// TIA Portal V16 export
// export: Created 2021-11-12T13:32:21.9335277Z, ExportSetting WithDefaults, DisplayName Totally Integrated Automation Portal, DisplayVersion V16 Update 3, DisplayName TIA Portal Version Control Interface, DisplayVersion V16 Update 2, DisplayName TIA Portal Openness, DisplayVersion V16 Update 3, DisplayName SINAMICS Startdrive Advanced, DisplayVersion V16 Update 5, DisplayName SINAMICS Startdrive G130, G150, S120, S150, SINAMICS MV, S210, DisplayVersion V16 Update 5, DisplayName SINAMICS Startdrive G110M, G120, G120C, G120D, G120P, G115D, DisplayVersion V16 Update 5, DisplayName STEP 7 Professional, DisplayVersion V16 Update 3, DisplayName STEP 7 Safety, DisplayVersion V16, DisplayName WinCC UA Professional, DisplayVersion V16 Update 3
FUNCTION_BLOCK "Station1R2"   // FB34, LAD
{ S7_Optimized_Access := 'TRUE' }
VERSION : 0.1
// stored: AutoNumber true, IsIECCheckEnabled false, IsRetainMemResEnabled false, MemoryReserve 100, SetENOAutomatically false, UDAEnableTagReadback false
   VAR
      SF_RO01_Timeout : "STD_DI_Mon";   // Move timeout
      "SF_CL01-BG01_Alarm" { S7_SetPoint := 'True'} : "STD_DI_Mon";
      "SF_CL01-BG02_Alarm" { S7_SetPoint := 'True'} : "STD_DI_Mon";
      SF_RC01 : "STD_DriveRobotABB";
      SF_RO01 : "STD_RobotABB";
      SF_RobotGripper : "STD_RobotGripper";
      SS_RobotZones { S7_SetPoint := 'True'} : "STD_RobotZones";
      SS_Edge { S7_SetPoint := 'True'} : Array[0..100] of Bool;
   END_VAR
   VAR RETAIN
      SDIPartID : DInt;
      SI_PartType : Int;
   END_VAR
   VAR
      SI_140RowNo : Int;   // Row number in map of station 140
      SI_140LineNo : Int;   // Line number in map of station 140
      SB1PutPosFound140 : Bool;   // Put position in map of station 140 found
      SB1ReqToChangeTool : Bool;   // Request from zone command to change tools
      SB1_1R2ChangeToolDone : Bool;   // Changing tool process done
      SB1_1R2GripperToTakeUp : Bool;
      SB1_1R2PutToolDone : Bool;
      SB1_1R1ToolSwitchDone : Bool;
      SB1CycleAutostop : Bool;   // Cycle autostop command
      SB1ServicePosReq { ExternalAccessible := 'False'; ExternalVisible := 'False'; ExternalWritable := 'False'} : Bool;   // Request to go to/from service position
      SB1RobotInitialized : Bool;   // Robot is initialized
   END_VAR
   VAR_TEMP
      TS_RC01 : "UDT_DriveRobotABBControl";   // Robot controller RC01 control
      TS_RO01 : "UDT_RobotABBControl";   // Robot RO01 control
      TI_RowNo : Int;
      TI_LineNo : Int;
      TB1PwrOK : Bool;   // Power for this station is OK
      TB1HomePosReq : Bool;   // Request to go to home position
      TB1Take120 : Bool;   // Take parts from 120
      TB1Put140 : Bool;   // Put parts to 140
      TB1CtrlRun : Bool;   // Robot controller is running in automat
      TB1GripperFree : Bool;
      TB1ChangeTool1R1UpDown : Bool;   // Change tool from upper possition
      TB1ChangeTool1R1DownUp : Bool;   // Change tool from lower possition
      TB1PutTool1R2Up : Bool;
      TB1PutTool1R2Down : Bool;
      TB1TakeTool1R2Up : Bool;
      TB1TakeTool1R2Down : Bool;
   END_VAR
   VAR CONSTANT
      CI_JobHome : UInt := 1;
      CI_JobService : UInt := 2;
      CI_JobPutToo1R2Up : UInt := 11;
      CI_JobPutToo1R2Down : UInt := 12;
      CI_JobChangeTool1R1UpDown : UInt := 21;
      CI_JobChangeTool1R1DownUp : UInt := 22;
      CI_JobTakeTool1R2Up : UInt := 31;
      CI_JobTakeTool1R2Down : UInt := 32;
      CI_JobTakeParts : UInt := 100;
      CI_JobPutPartsPos11 : UInt := 201;
      CI_JobPutPartsPos15 : UInt := 202;
      CI_JobPutPartsPos19 : UInt := 203;
      CI_JobPutPartsPos21 : UInt := 204;
      CI_JobPutPartsPos25 : UInt := 205;
      CI_JobPutPartsPos29 : UInt := 206;
   END_VAR
   VAR_TEMP   // added for the SCL form of the ladder/FBD networks
      _w1 : Bool;
      _w2 : Bool;
      _w3 : Bool;
      _w4 : Bool;
      _w5 : Bool;
      _w6 : Bool;
      _w7 : Bool;
      _w8 : Bool;
   END_VAR
BEGIN

REGION Network 1: Clear temporary variables
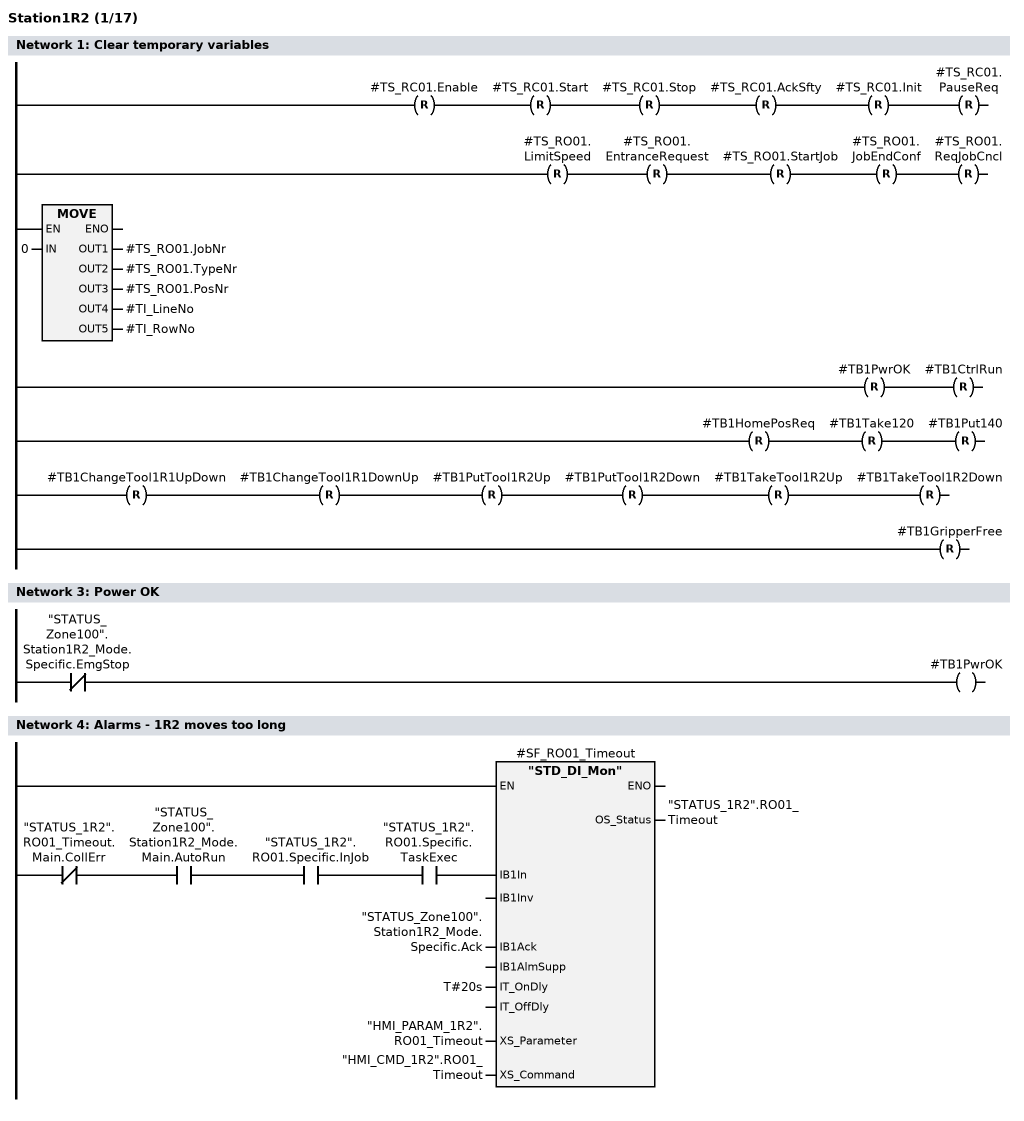
   RUNG wire#powerrail
      R_Coil( #TS_RC01.Enable )
      R_Coil( #TS_RC01.Start )
      R_Coil( #TS_RC01.Stop )
      R_Coil( #TS_RC01.AckSfty )
      R_Coil( #TS_RC01.Init )
      R_Coil( #TS_RC01.PauseReq )
   END_RUNG
   RUNG wire#powerrail
      R_Coil( #TS_RO01.LimitSpeed )
      R_Coil( #TS_RO01.EntranceRequest )
      R_Coil( #TS_RO01.StartJob )
      R_Coil( #TS_RO01.JobEndConf )
      R_Coil( #TS_RO01.ReqJobCncl )
   END_RUNG
   RUNG wire#powerrail
      Move(in := 0, out1 => #TS_RO01.JobNr, out2 => #TS_RO01.TypeNr, out3 => #TS_RO01.PosNr, out4 => #TI_LineNo, out5 => #TI_RowNo)
   END_RUNG
   RUNG wire#powerrail
      R_Coil( #TB1PwrOK )
      R_Coil( #TB1CtrlRun )
   END_RUNG
   RUNG wire#powerrail
      R_Coil( #TB1HomePosReq )
      R_Coil( #TB1Take120 )
      R_Coil( #TB1Put140 )
   END_RUNG
   RUNG wire#powerrail
      R_Coil( #TB1ChangeTool1R1UpDown )
      R_Coil( #TB1ChangeTool1R1DownUp )
      R_Coil( #TB1PutTool1R2Up )
      R_Coil( #TB1PutTool1R2Down )
      R_Coil( #TB1TakeTool1R2Up )
      R_Coil( #TB1TakeTool1R2Down )
   END_RUNG
   RUNG wire#powerrail
      R_Coil( #TB1GripperFree )
   END_RUNG
   // the same network as SCL:
   #TS_RC01.Enable := FALSE;
   #TS_RC01.Start := FALSE;
   #TS_RC01.Stop := FALSE;
   #TS_RC01.AckSfty := FALSE;
   #TS_RC01.Init := FALSE;
   #TS_RC01.PauseReq := FALSE;
   #TS_RO01.LimitSpeed := FALSE;
   #TS_RO01.EntranceRequest := FALSE;
   #TS_RO01.StartJob := FALSE;
   #TS_RO01.JobEndConf := FALSE;
   #TS_RO01.ReqJobCncl := FALSE;
   #TS_RO01.JobNr := 0;
   #TS_RO01.TypeNr := 0;
   #TS_RO01.PosNr := 0;
   #TI_LineNo := 0;
   #TI_RowNo := 0;
   #TB1PwrOK := FALSE;
   #TB1CtrlRun := FALSE;
   #TB1HomePosReq := FALSE;
   #TB1Take120 := FALSE;
   #TB1Put140 := FALSE;
   #TB1ChangeTool1R1UpDown := FALSE;
   #TB1ChangeTool1R1DownUp := FALSE;
   #TB1PutTool1R2Up := FALSE;
   #TB1PutTool1R2Down := FALSE;
   #TB1TakeTool1R2Up := FALSE;
   #TB1TakeTool1R2Down := FALSE;
   #TB1GripperFree := FALSE;
END_REGION

REGION Network 2: *************** Alarms ***************
END_REGION

REGION Network 3: Power OK
   RUNG wire#powerrail
      I_Contact( "STATUS_Zone100".Station1R2_Mode.Specific.EmgStop )
      Coil( #TB1PwrOK )
   END_RUNG
   // the same network as SCL:
   #TB1PwrOK := NOT "STATUS_Zone100".Station1R2_Mode.Specific.EmgStop;
END_REGION

REGION Network 4: Alarms - 1R2 moves too long
   RUNG wire#powerrail
      #SF_RO01_Timeout(IB1In := wire#w1, IB1Inv :=, IB1Ack := "STATUS_Zone100".Station1R2_Mode.Specific.Ack, IB1AlmSupp :=, IT_OnDly := T#20s, IT_OffDly :=, XS_Parameter := "HMI_PARAM_1R2".RO01_Timeout, XS_Command := "HMI_CMD_1R2".RO01_Timeout, OS_Status => "STATUS_1R2".RO01_Timeout)
   END_RUNG
   RUNG wire#powerrail
      I_Contact( "STATUS_1R2".RO01_Timeout.Main.CollErr )
      Contact( "STATUS_Zone100".Station1R2_Mode.Main.AutoRun )
      Contact( "STATUS_1R2".RO01.Specific.InJob )
      Contact( "STATUS_1R2".RO01.Specific.TaskExec )
   END_RUNG wire#w1
   // the same network as SCL:
   #SF_RO01_Timeout(IB1In := NOT "STATUS_1R2".RO01_Timeout.Main.CollErr AND "STATUS_Zone100".Station1R2_Mode.Main.AutoRun AND "STATUS_1R2".RO01.Specific.InJob AND "STATUS_1R2".RO01.Specific.TaskExec,   // "STD_DI_Mon"
                    IB1Ack := "STATUS_Zone100".Station1R2_Mode.Specific.Ack,
                    IT_OnDly := T#20s,
                    XS_Parameter := "HMI_PARAM_1R2".RO01_Timeout,
                    XS_Command := "HMI_CMD_1R2".RO01_Timeout,
                    OS_Status => "STATUS_1R2".RO01_Timeout);
END_REGION

REGION Network 5: Sensor alarms - CL01
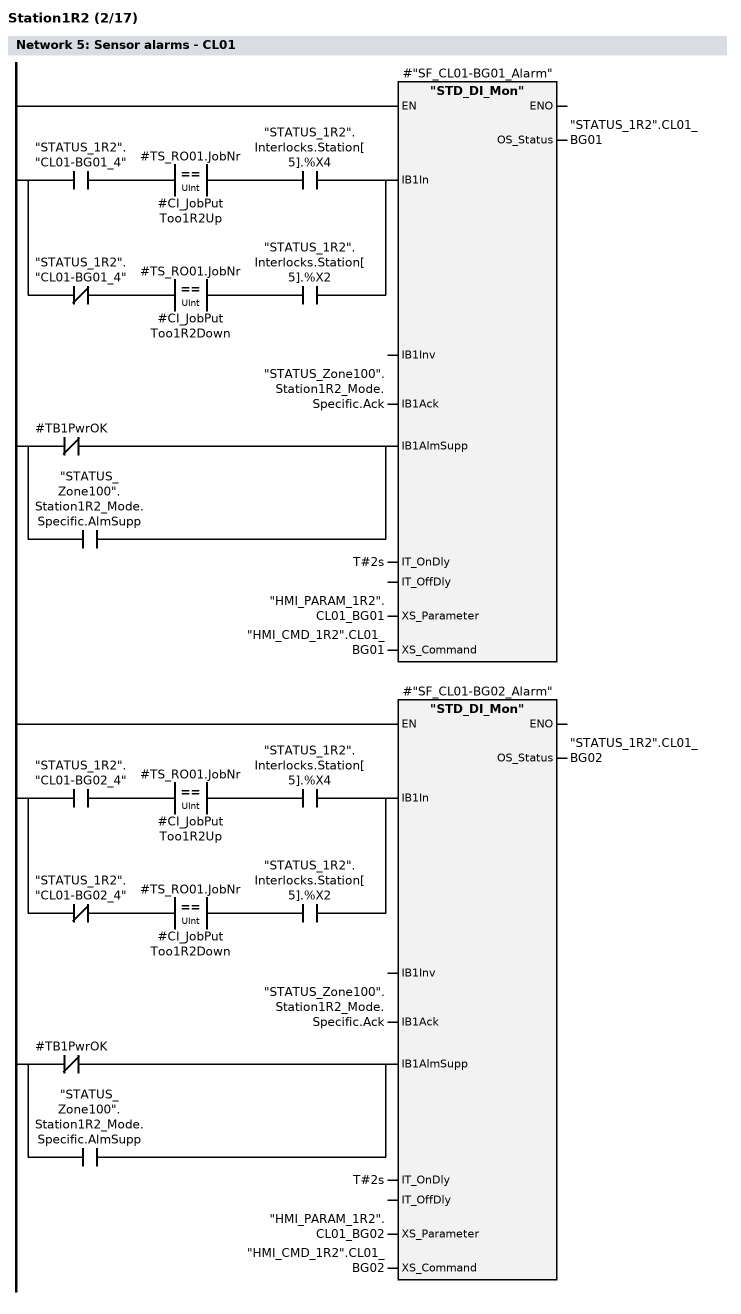
   RUNG wire#powerrail
      #"SF_CL01-BG01_Alarm"(IB1In := wire#w1, IB1AlmSupp := wire#w2, IB1Inv :=, IB1Ack := "STATUS_Zone100".Station1R2_Mode.Specific.Ack, IT_OnDly := T#2s, IT_OffDly :=, XS_Parameter := "HMI_PARAM_1R2".CL01_BG01, XS_Command := "HMI_CMD_1R2".CL01_BG01, OS_Status => "STATUS_1R2".CL01_BG01)
   END_RUNG
   RUNG wire#powerrail
      Contact( "STATUS_1R2"."CL01-BG01_4" )
      { S7_Templates := "SrcType := UInt" } EQ_Contact(in1 := #TS_RO01.JobNr, in2 := #CI_JobPutToo1R2Up)
      Contact( "STATUS_1R2".Interlocks.Station[5].%X4 )
   END_RUNG wire#w1
   RUNG wire#powerrail
      I_Contact( "STATUS_1R2"."CL01-BG01_4" )
      { S7_Templates := "SrcType := UInt" } EQ_Contact(in1 := #TS_RO01.JobNr, in2 := #CI_JobPutToo1R2Down)
      Contact( "STATUS_1R2".Interlocks.Station[5].%X2 )
   END_RUNG wire#w1
   RUNG wire#powerrail
      I_Contact( #TB1PwrOK )
   END_RUNG wire#w2
   RUNG wire#powerrail
      Contact( "STATUS_Zone100".Station1R2_Mode.Specific.AlmSupp )
   END_RUNG wire#w2
   RUNG wire#powerrail
      #"SF_CL01-BG02_Alarm"(IB1In := wire#w3, IB1AlmSupp := wire#w4, IB1Inv :=, IB1Ack := "STATUS_Zone100".Station1R2_Mode.Specific.Ack, IT_OnDly := T#2s, IT_OffDly :=, XS_Parameter := "HMI_PARAM_1R2".CL01_BG02, XS_Command := "HMI_CMD_1R2".CL01_BG02, OS_Status => "STATUS_1R2".CL01_BG02)
   END_RUNG
   RUNG wire#powerrail
      Contact( "STATUS_1R2"."CL01-BG02_4" )
      { S7_Templates := "SrcType := UInt" } EQ_Contact(in1 := #TS_RO01.JobNr, in2 := #CI_JobPutToo1R2Up)
      Contact( "STATUS_1R2".Interlocks.Station[5].%X4 )
   END_RUNG wire#w3
   RUNG wire#powerrail
      I_Contact( "STATUS_1R2"."CL01-BG02_4" )
      { S7_Templates := "SrcType := UInt" } EQ_Contact(in1 := #TS_RO01.JobNr, in2 := #CI_JobPutToo1R2Down)
      Contact( "STATUS_1R2".Interlocks.Station[5].%X2 )
   END_RUNG wire#w3
   RUNG wire#powerrail
      I_Contact( #TB1PwrOK )
   END_RUNG wire#w4
   RUNG wire#powerrail
      Contact( "STATUS_Zone100".Station1R2_Mode.Specific.AlmSupp )
   END_RUNG wire#w4
   // the same network as SCL:
   #"SF_CL01-BG01_Alarm"(IB1In := ("STATUS_1R2"."CL01-BG01_4" AND (#TS_RO01.JobNr = #CI_JobPutToo1R2Up) AND "STATUS_1R2".Interlocks.Station[5].%X4) OR (NOT "STATUS_1R2"."CL01-BG01_4" AND (#TS_RO01.JobNr = #CI_JobPutToo1R2Down) AND "STATUS_1R2".Interlocks.Station[5].%X2),   // "STD_DI_Mon"
                         IB1Ack := "STATUS_Zone100".Station1R2_Mode.Specific.Ack,
                         IB1AlmSupp := NOT #TB1PwrOK OR "STATUS_Zone100".Station1R2_Mode.Specific.AlmSupp,
                         IT_OnDly := T#2s,
                         XS_Parameter := "HMI_PARAM_1R2".CL01_BG01,
                         XS_Command := "HMI_CMD_1R2".CL01_BG01,
                         OS_Status => "STATUS_1R2".CL01_BG01);
   #"SF_CL01-BG02_Alarm"(IB1In := ("STATUS_1R2"."CL01-BG02_4" AND (#TS_RO01.JobNr = #CI_JobPutToo1R2Up) AND "STATUS_1R2".Interlocks.Station[5].%X4) OR (NOT "STATUS_1R2"."CL01-BG02_4" AND (#TS_RO01.JobNr = #CI_JobPutToo1R2Down) AND "STATUS_1R2".Interlocks.Station[5].%X2),   // "STD_DI_Mon"
                         IB1Ack := "STATUS_Zone100".Station1R2_Mode.Specific.Ack,
                         IB1AlmSupp := NOT #TB1PwrOK OR "STATUS_Zone100".Station1R2_Mode.Specific.AlmSupp,
                         IT_OnDly := T#2s,
                         XS_Parameter := "HMI_PARAM_1R2".CL01_BG02,
                         XS_Command := "HMI_CMD_1R2".CL01_BG02,
                         OS_Status => "STATUS_1R2".CL01_BG02);
END_REGION

REGION Network 6: *************** Controller RC01 ***************
END_REGION

REGION Network 7: Controller RC01 - control
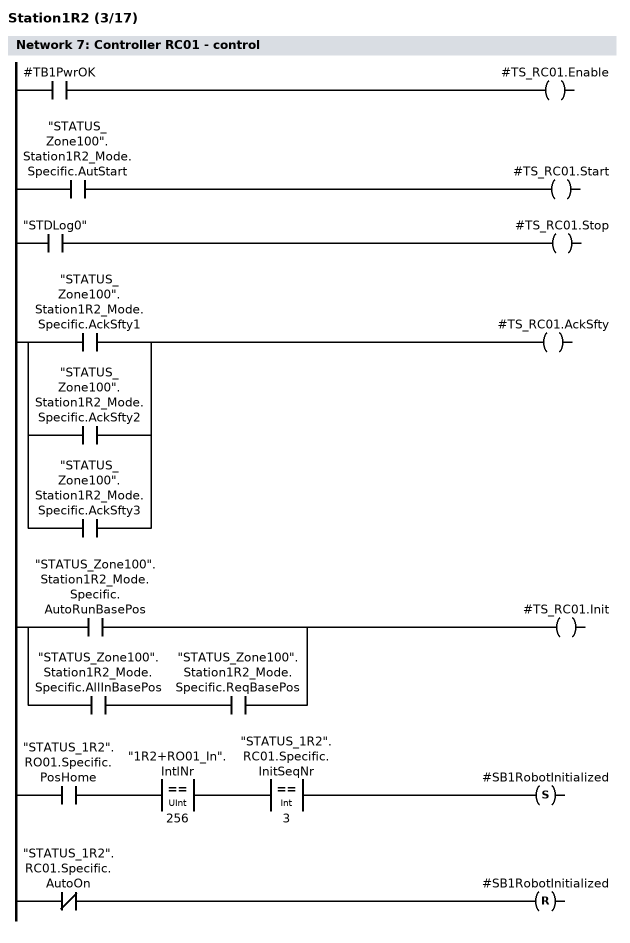
   RUNG wire#powerrail
      Contact( #TB1PwrOK )
      Coil( #TS_RC01.Enable )
   END_RUNG
   RUNG wire#powerrail
      Contact( "STATUS_Zone100".Station1R2_Mode.Specific.AutStart )
      Coil( #TS_RC01.Start )
   END_RUNG
   RUNG wire#powerrail
      Contact( "STDLog0" )
      Coil( #TS_RC01.Stop )
   END_RUNG
   RUNG wire#powerrail
      Contact( "STATUS_Zone100".Station1R2_Mode.Specific.AckSfty1 )
      wire#w1
      Coil( #TS_RC01.AckSfty )
   END_RUNG
   RUNG wire#powerrail
      Contact( "STATUS_Zone100".Station1R2_Mode.Specific.AckSfty2 )
   END_RUNG wire#w1
   RUNG wire#powerrail
      Contact( "STATUS_Zone100".Station1R2_Mode.Specific.AckSfty3 )
   END_RUNG wire#w1
   RUNG wire#powerrail
      Contact( "STATUS_Zone100".Station1R2_Mode.Specific.AutoRunBasePos )
      wire#w2
      Coil( #TS_RC01.Init )
   END_RUNG
   RUNG wire#powerrail
      Contact( "STATUS_Zone100".Station1R2_Mode.Specific.AllInBasePos )
      Contact( "STATUS_Zone100".Station1R2_Mode.Specific.ReqBasePos )
   END_RUNG wire#w2
   RUNG wire#powerrail
      Contact( "STATUS_1R2".RO01.Specific.PosHome )
      { S7_Templates := "SrcType := UInt" } EQ_Contact(in1 := "1R2+RO01_In".IntlNr, in2 := 256)
      { S7_Templates := "SrcType := Int" } EQ_Contact(in1 := "STATUS_1R2".RC01.Specific.InitSeqNr, in2 := 3)
      S_Coil( #SB1RobotInitialized )
   END_RUNG
   RUNG wire#powerrail
      I_Contact( "STATUS_1R2".RC01.Specific.AutoOn )
      R_Coil( #SB1RobotInitialized )
   END_RUNG
   // the same network as SCL:
   #TS_RC01.Enable := #TB1PwrOK;
   #TS_RC01.Start := "STATUS_Zone100".Station1R2_Mode.Specific.AutStart;
   #TS_RC01.Stop := "STDLog0";
   #TS_RC01.AckSfty := "STATUS_Zone100".Station1R2_Mode.Specific.AckSfty1 OR "STATUS_Zone100".Station1R2_Mode.Specific.AckSfty2 OR "STATUS_Zone100".Station1R2_Mode.Specific.AckSfty3;
   #TS_RC01.Init := "STATUS_Zone100".Station1R2_Mode.Specific.AutoRunBasePos OR ("STATUS_Zone100".Station1R2_Mode.Specific.AllInBasePos AND "STATUS_Zone100".Station1R2_Mode.Specific.ReqBasePos);
   IF "STATUS_1R2".RO01.Specific.PosHome AND ("1R2+RO01_In".IntlNr = 256) AND ("STATUS_1R2".RC01.Specific.InitSeqNr = 3) THEN
       #SB1RobotInitialized := TRUE;
   END_IF;
   IF NOT "STATUS_1R2".RC01.Specific.AutoOn THEN #SB1RobotInitialized := FALSE; END_IF;
END_REGION

REGION Network 8: Controller RC01 - request to pause robots jobs
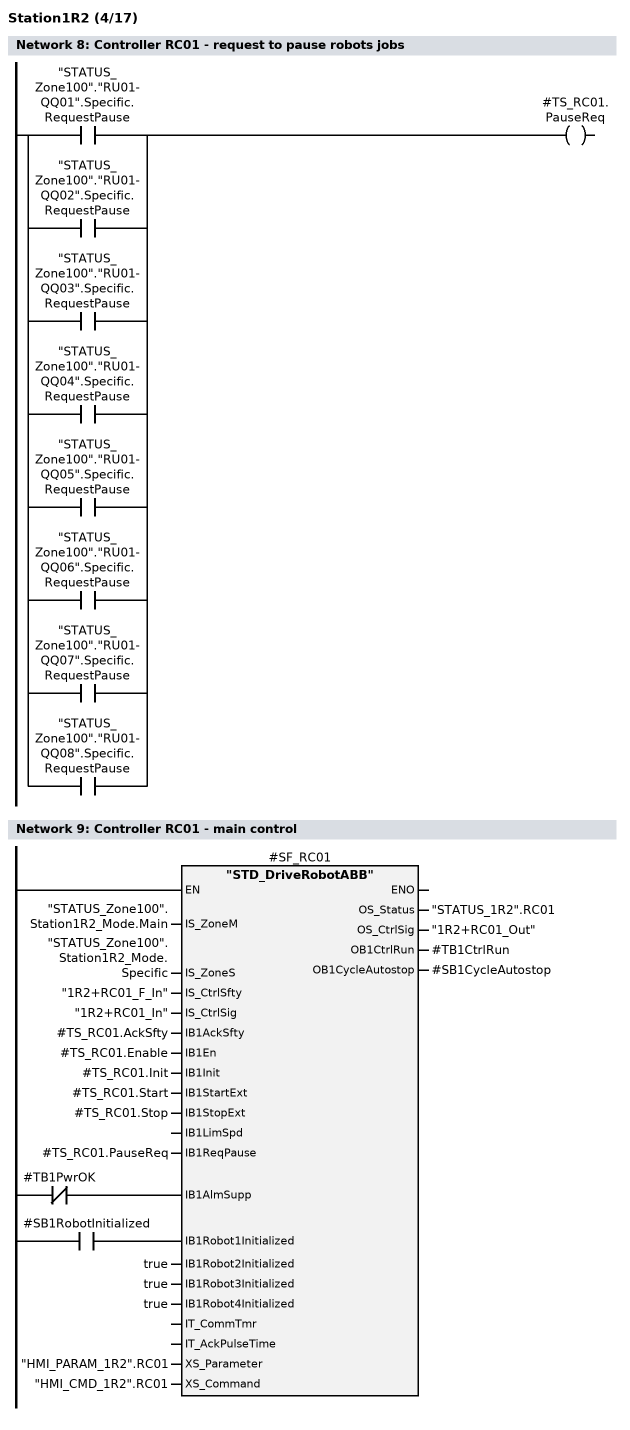
   RUNG wire#powerrail
      Contact( "STATUS_Zone100"."RU01-QQ01".Specific.RequestPause )
      wire#w1
      Coil( #TS_RC01.PauseReq )
   END_RUNG
   RUNG wire#powerrail
      Contact( "STATUS_Zone100"."RU01-QQ02".Specific.RequestPause )
   END_RUNG wire#w1
   RUNG wire#powerrail
      Contact( "STATUS_Zone100"."RU01-QQ03".Specific.RequestPause )
   END_RUNG wire#w1
   RUNG wire#powerrail
      Contact( "STATUS_Zone100"."RU01-QQ04".Specific.RequestPause )
   END_RUNG wire#w1
   RUNG wire#powerrail
      Contact( "STATUS_Zone100"."RU01-QQ05".Specific.RequestPause )
   END_RUNG wire#w1
   RUNG wire#powerrail
      Contact( "STATUS_Zone100"."RU01-QQ06".Specific.RequestPause )
   END_RUNG wire#w1
   RUNG wire#powerrail
      Contact( "STATUS_Zone100"."RU01-QQ07".Specific.RequestPause )
   END_RUNG wire#w1
   RUNG wire#powerrail
      Contact( "STATUS_Zone100"."RU01-QQ08".Specific.RequestPause )
   END_RUNG wire#w1
   // the same network as SCL:
   #TS_RC01.PauseReq := "STATUS_Zone100"."RU01-QQ01".Specific.RequestPause OR "STATUS_Zone100"."RU01-QQ02".Specific.RequestPause OR "STATUS_Zone100"."RU01-QQ03".Specific.RequestPause OR "STATUS_Zone100"."RU01-QQ04".Specific.RequestPause OR "STATUS_Zone100"."RU01-QQ05".Specific.RequestPause OR "STATUS_Zone100"."RU01-QQ06".Specific.RequestPause OR "STATUS_Zone100"."RU01-QQ07".Specific.RequestPause OR "STATUS_Zone100"."RU01-QQ08".Specific.RequestPause;
END_REGION

REGION Network 9: Controller RC01 - main control
   RUNG wire#powerrail
      #SF_RC01(IB1AlmSupp := wire#w1, IB1Robot1Initialized := wire#w2, IS_ZoneM := "STATUS_Zone100".Station1R2_Mode.Main, IS_ZoneS := "STATUS_Zone100".Station1R2_Mode.Specific, IS_CtrlSfty := "1R2+RC01_F_In", IS_CtrlSig := "1R2+RC01_In", IB1AckSfty := #TS_RC01.AckSfty, IB1En := #TS_RC01.Enable, IB1Init := #TS_RC01.Init, IB1StartExt := #TS_RC01.Start, IB1StopExt := #TS_RC01.Stop, IB1LimSpd :=, IB1ReqPause := #TS_RC01.PauseReq, IB1Robot2Initialized := true, IB1Robot3Initialized := true, IB1Robot4Initialized := true, IT_CommTmr :=, IT_AckPulseTime :=, XS_Parameter := "HMI_PARAM_1R2".RC01, XS_Command := "HMI_CMD_1R2".RC01, OS_Status => "STATUS_1R2".RC01, OS_CtrlSig => "1R2+RC01_Out", OB1CtrlRun => #TB1CtrlRun, OB1CycleAutostop => #SB1CycleAutostop)
   END_RUNG
   RUNG wire#powerrail
      I_Contact( #TB1PwrOK )
   END_RUNG wire#w1
   RUNG wire#powerrail
      Contact( #SB1RobotInitialized )
   END_RUNG wire#w2
   // the same network as SCL:
   #SF_RC01(IS_ZoneM := "STATUS_Zone100".Station1R2_Mode.Main,   // "STD_DriveRobotABB"
            IS_ZoneS := "STATUS_Zone100".Station1R2_Mode.Specific,
            IS_CtrlSfty := "1R2+RC01_F_In",
            IS_CtrlSig := "1R2+RC01_In",
            IB1AckSfty := #TS_RC01.AckSfty,
            IB1En := #TS_RC01.Enable,
            IB1Init := #TS_RC01.Init,
            IB1StartExt := #TS_RC01.Start,
            IB1StopExt := #TS_RC01.Stop,
            IB1ReqPause := #TS_RC01.PauseReq,
            IB1AlmSupp := NOT #TB1PwrOK,
            IB1Robot1Initialized := #SB1RobotInitialized,
            IB1Robot2Initialized := true,
            IB1Robot3Initialized := true,
            IB1Robot4Initialized := true,
            XS_Parameter := "HMI_PARAM_1R2".RC01,
            XS_Command := "HMI_CMD_1R2".RC01,
            OS_Status => "STATUS_1R2".RC01,
            OS_CtrlSig => "1R2+RC01_Out",
            OB1CtrlRun => #TB1CtrlRun,
            OB1CycleAutostop => #SB1CycleAutostop);
END_REGION

REGION Network 10: *************** Robot RO01 ***************
END_REGION

REGION Network 11: Robot RO01 - speed limit
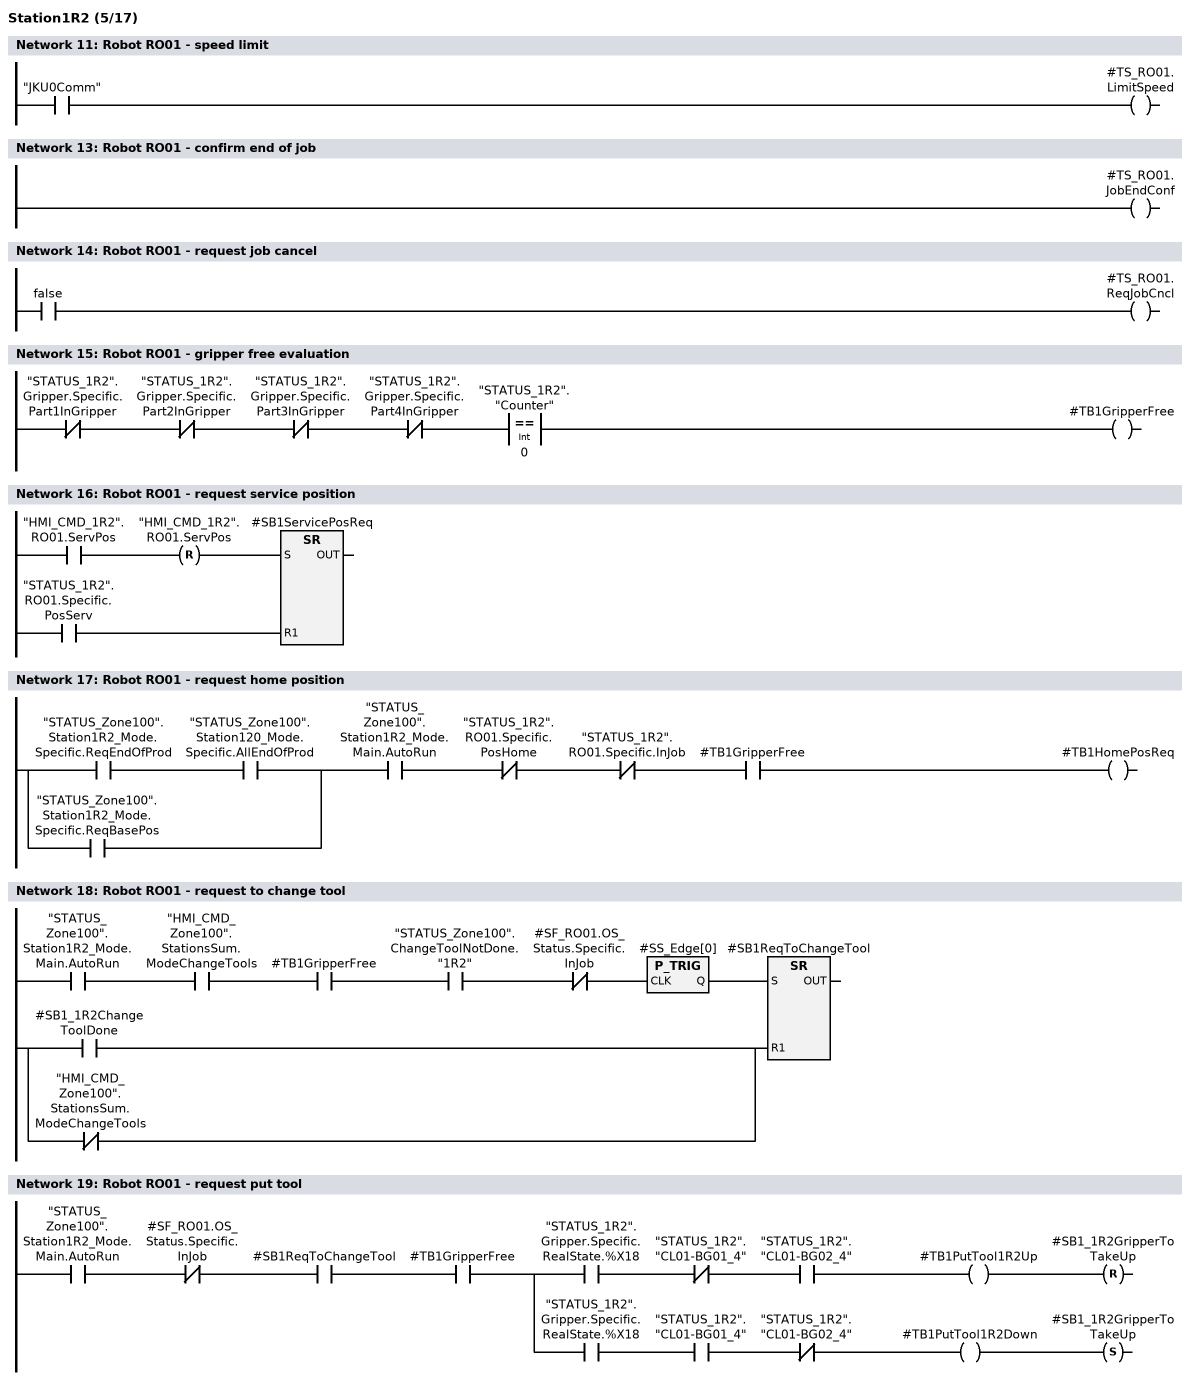
   RUNG wire#powerrail
      Contact( "JKU0Comm" )
      Coil( #TS_RO01.LimitSpeed )
   END_RUNG
   // the same network as SCL:
   #TS_RO01.LimitSpeed := "JKU0Comm";
END_REGION

REGION Network 12: Robot RO01 - position number
END_REGION

REGION Network 13: Robot RO01 - confirm end of job
   RUNG wire#powerrail
      Coil( #TS_RO01.JobEndConf )
   END_RUNG
   // the same network as SCL:
   #TS_RO01.JobEndConf := TRUE;
END_REGION

REGION Network 14: Robot RO01 - request job cancel
   RUNG wire#powerrail
      Contact( false )
      Coil( #TS_RO01.ReqJobCncl )
   END_RUNG
   // the same network as SCL:
   #TS_RO01.ReqJobCncl := false;
END_REGION

REGION Network 15: Robot RO01 - gripper free evaluation
   RUNG wire#powerrail
      I_Contact( "STATUS_1R2".Gripper.Specific.Part1InGripper )
      I_Contact( "STATUS_1R2".Gripper.Specific.Part2InGripper )
      I_Contact( "STATUS_1R2".Gripper.Specific.Part3InGripper )
      I_Contact( "STATUS_1R2".Gripper.Specific.Part4InGripper )
      { S7_Templates := "SrcType := Int" } EQ_Contact(in1 := "STATUS_1R2"."Counter", in2 := 0)
      Coil( #TB1GripperFree )
   END_RUNG
   // the same network as SCL:
   #TB1GripperFree := NOT "STATUS_1R2".Gripper.Specific.Part1InGripper AND NOT "STATUS_1R2".Gripper.Specific.Part2InGripper AND NOT "STATUS_1R2".Gripper.Specific.Part3InGripper AND NOT "STATUS_1R2".Gripper.Specific.Part4InGripper AND ("STATUS_1R2"."Counter" = 0);
END_REGION

REGION Network 16: Robot RO01 - request service position
   RUNG wire#powerrail
      Contact( "HMI_CMD_1R2".RO01.ServPos )
      R_Coil( "HMI_CMD_1R2".RO01.ServPos )
      S_SR(operand := #SB1ServicePosReq, r1 := wire#w1)
   END_RUNG
   RUNG wire#powerrail
      Contact( "STATUS_1R2".RO01.Specific.PosServ )
   END_RUNG wire#w1
   // the same network as SCL:
   #_w1 := "HMI_CMD_1R2".RO01.ServPos;
   IF #_w1 THEN
       "HMI_CMD_1R2".RO01.ServPos := FALSE;
       #SB1ServicePosReq := TRUE;   // SR flip-flop
   END_IF;
   IF "STATUS_1R2".RO01.Specific.PosServ THEN #SB1ServicePosReq := FALSE; END_IF;
END_REGION

REGION Network 17: Robot RO01 - request home position
   RUNG wire#powerrail
      Contact( "STATUS_Zone100".Station1R2_Mode.Specific.ReqEndOfProd )
      Contact( "STATUS_Zone100".Station120_Mode.Specific.AllEndOfProd )
      wire#w1
      Contact( "STATUS_Zone100".Station1R2_Mode.Main.AutoRun )
      I_Contact( "STATUS_1R2".RO01.Specific.PosHome )
      I_Contact( "STATUS_1R2".RO01.Specific.InJob )
      Contact( #TB1GripperFree )
      Coil( #TB1HomePosReq )
   END_RUNG
   RUNG wire#powerrail
      Contact( "STATUS_Zone100".Station1R2_Mode.Specific.ReqBasePos )
   END_RUNG wire#w1
   // the same network as SCL:
   #TB1HomePosReq := (("STATUS_Zone100".Station1R2_Mode.Specific.ReqEndOfProd AND "STATUS_Zone100".Station120_Mode.Specific.AllEndOfProd) OR "STATUS_Zone100".Station1R2_Mode.Specific.ReqBasePos) AND "STATUS_Zone100".Station1R2_Mode.Main.AutoRun AND NOT "STATUS_1R2".RO01.Specific.PosHome AND NOT "STATUS_1R2".RO01.Specific.InJob AND #TB1GripperFree;
END_REGION

REGION Network 18: Robot RO01 - request to change tool
   RUNG wire#powerrail
      Contact( "STATUS_Zone100".Station1R2_Mode.Main.AutoRun )
      Contact( "HMI_CMD_Zone100".StationsSum.ModeChangeTools )
      Contact( #TB1GripperFree )
      Contact( "STATUS_Zone100".ChangeToolNotDone."1R2" )
      I_Contact( #SF_RO01.OS_Status.Specific.InJob )
      P_Trig( #SS_Edge[0] )
      S_SR(operand := #SB1ReqToChangeTool, r1 := wire#w1)
   END_RUNG
   RUNG wire#powerrail
      Contact( #SB1_1R2ChangeToolDone )
   END_RUNG wire#w1
   RUNG wire#powerrail
      I_Contact( "HMI_CMD_Zone100".StationsSum.ModeChangeTools )
   END_RUNG wire#w1
   // the same network as SCL:
   #_w1 := "STATUS_Zone100".Station1R2_Mode.Main.AutoRun AND "HMI_CMD_Zone100".StationsSum.ModeChangeTools AND #TB1GripperFree AND "STATUS_Zone100".ChangeToolNotDone."1R2" AND NOT #SF_RO01.OS_Status.Specific.InJob;
   #_w2 := #_w1 AND NOT #SS_Edge[0];   // rising edge
   #SS_Edge[0] := #_w1;
   IF #_w2 THEN
       #SB1ReqToChangeTool := TRUE;   // SR flip-flop
   END_IF;
   IF #SB1_1R2ChangeToolDone OR NOT "HMI_CMD_Zone100".StationsSum.ModeChangeTools THEN
       #SB1ReqToChangeTool := FALSE;
   END_IF;
END_REGION

REGION Network 19: Robot RO01 - request put tool
   RUNG wire#powerrail
      Contact( "STATUS_Zone100".Station1R2_Mode.Main.AutoRun )
      I_Contact( #SF_RO01.OS_Status.Specific.InJob )
      Contact( #SB1ReqToChangeTool )
      Contact( #TB1GripperFree )
      wire#w1
      Contact( "STATUS_1R2".Gripper.Specific.RealState.%X18 )
      I_Contact( "STATUS_1R2"."CL01-BG01_4" )
      Contact( "STATUS_1R2"."CL01-BG02_4" )
      Coil( #TB1PutTool1R2Up )
      R_Coil( #SB1_1R2GripperToTakeUp )
   END_RUNG
   RUNG wire#w1
      Contact( "STATUS_1R2".Gripper.Specific.RealState.%X18 )
      Contact( "STATUS_1R2"."CL01-BG01_4" )
      I_Contact( "STATUS_1R2"."CL01-BG02_4" )
      Coil( #TB1PutTool1R2Down )
      S_Coil( #SB1_1R2GripperToTakeUp )
   END_RUNG
   // the same network as SCL:
   #_w1 := "STATUS_Zone100".Station1R2_Mode.Main.AutoRun AND NOT #SF_RO01.OS_Status.Specific.InJob AND #SB1ReqToChangeTool AND #TB1GripperFree;
   #TB1PutTool1R2Up := #_w1 AND "STATUS_1R2".Gripper.Specific.RealState.%X18 AND NOT "STATUS_1R2"."CL01-BG01_4" AND "STATUS_1R2"."CL01-BG02_4";
   IF #TB1PutTool1R2Up THEN #SB1_1R2GripperToTakeUp := FALSE; END_IF;
   #TB1PutTool1R2Down := #_w1 AND "STATUS_1R2".Gripper.Specific.RealState.%X18 AND "STATUS_1R2"."CL01-BG01_4" AND NOT "STATUS_1R2"."CL01-BG02_4";
   IF #TB1PutTool1R2Down THEN #SB1_1R2GripperToTakeUp := TRUE; END_IF;
END_REGION

REGION Network 20: Robot Ro01 - change tool for 1R1
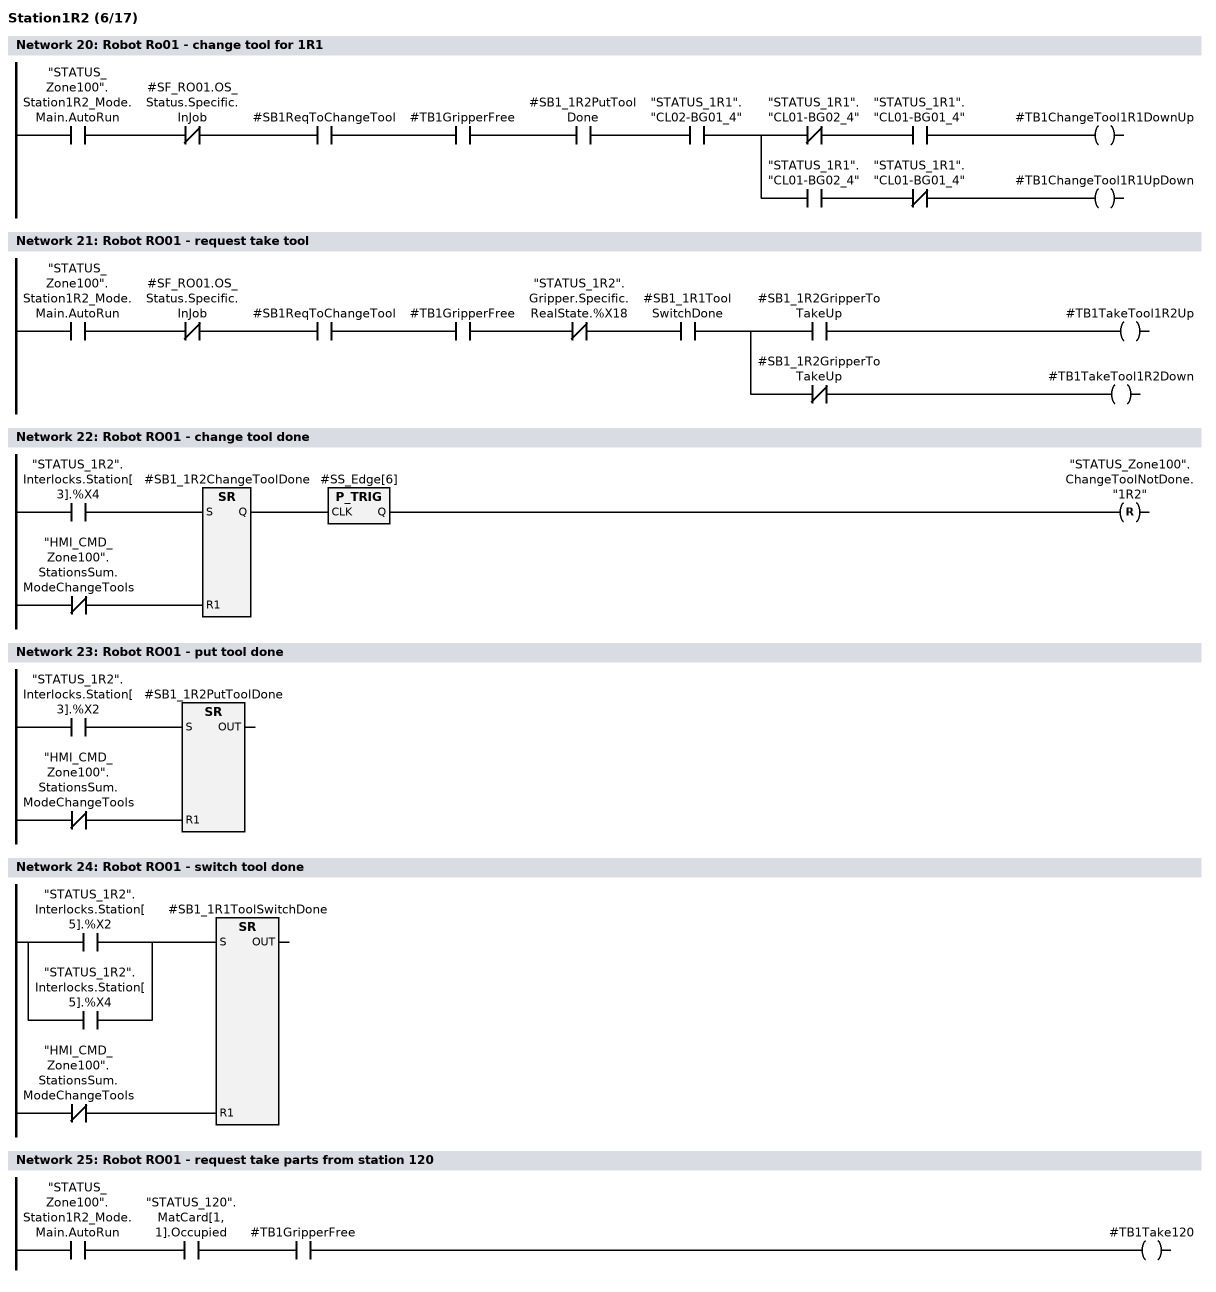
   RUNG wire#powerrail
      Contact( "STATUS_Zone100".Station1R2_Mode.Main.AutoRun )
      I_Contact( #SF_RO01.OS_Status.Specific.InJob )
      Contact( #SB1ReqToChangeTool )
      Contact( #TB1GripperFree )
      Contact( #SB1_1R2PutToolDone )
      Contact( "STATUS_1R1"."CL02-BG01_4" )
      wire#w1
      I_Contact( "STATUS_1R1"."CL01-BG02_4" )
      Contact( "STATUS_1R1"."CL01-BG01_4" )
      Coil( #TB1ChangeTool1R1DownUp )
   END_RUNG
   RUNG wire#w1
      Contact( "STATUS_1R1"."CL01-BG02_4" )
      I_Contact( "STATUS_1R1"."CL01-BG01_4" )
      Coil( #TB1ChangeTool1R1UpDown )
   END_RUNG
   // the same network as SCL:
   #_w1 := "STATUS_Zone100".Station1R2_Mode.Main.AutoRun AND NOT #SF_RO01.OS_Status.Specific.InJob AND #SB1ReqToChangeTool AND #TB1GripperFree AND #SB1_1R2PutToolDone AND "STATUS_1R1"."CL02-BG01_4";
   #TB1ChangeTool1R1DownUp := #_w1 AND NOT "STATUS_1R1"."CL01-BG02_4" AND "STATUS_1R1"."CL01-BG01_4";
   #TB1ChangeTool1R1UpDown := #_w1 AND "STATUS_1R1"."CL01-BG02_4" AND NOT "STATUS_1R1"."CL01-BG01_4";
END_REGION

REGION Network 21: Robot RO01 - request take tool
   RUNG wire#powerrail
      Contact( "STATUS_Zone100".Station1R2_Mode.Main.AutoRun )
      I_Contact( #SF_RO01.OS_Status.Specific.InJob )
      Contact( #SB1ReqToChangeTool )
      Contact( #TB1GripperFree )
      I_Contact( "STATUS_1R2".Gripper.Specific.RealState.%X18 )
      Contact( #SB1_1R1ToolSwitchDone )
      wire#w1
      Contact( #SB1_1R2GripperToTakeUp )
      Coil( #TB1TakeTool1R2Up )
   END_RUNG
   RUNG wire#w1
      I_Contact( #SB1_1R2GripperToTakeUp )
      Coil( #TB1TakeTool1R2Down )
   END_RUNG
   // the same network as SCL:
   #_w1 := "STATUS_Zone100".Station1R2_Mode.Main.AutoRun AND NOT #SF_RO01.OS_Status.Specific.InJob AND #SB1ReqToChangeTool AND #TB1GripperFree AND NOT "STATUS_1R2".Gripper.Specific.RealState.%X18 AND #SB1_1R1ToolSwitchDone;
   #TB1TakeTool1R2Up := #_w1 AND #SB1_1R2GripperToTakeUp;
   #TB1TakeTool1R2Down := #_w1 AND NOT #SB1_1R2GripperToTakeUp;
END_REGION

REGION Network 22: Robot RO01 - change tool done
   RUNG wire#powerrail
      Contact( "STATUS_1R2".Interlocks.Station[3].%X4 )
      S_SR(operand := #SB1_1R2ChangeToolDone, r1 := wire#w1)
      P_Trig( #SS_Edge[6] )
      R_Coil( "STATUS_Zone100".ChangeToolNotDone."1R2" )
   END_RUNG
   RUNG wire#powerrail
      I_Contact( "HMI_CMD_Zone100".StationsSum.ModeChangeTools )
   END_RUNG wire#w1
   // the same network as SCL:
   IF "STATUS_1R2".Interlocks.Station[3].%X4 THEN
       #SB1_1R2ChangeToolDone := TRUE;   // SR flip-flop
   END_IF;
   IF NOT "HMI_CMD_Zone100".StationsSum.ModeChangeTools THEN #SB1_1R2ChangeToolDone := FALSE; END_IF;
   #_w1 := #SB1_1R2ChangeToolDone AND NOT #SS_Edge[6];   // rising edge
   #SS_Edge[6] := #SB1_1R2ChangeToolDone;
   IF #_w1 THEN "STATUS_Zone100".ChangeToolNotDone."1R2" := FALSE; END_IF;
END_REGION

REGION Network 23: Robot RO01 - put tool done
   RUNG wire#powerrail
      Contact( "STATUS_1R2".Interlocks.Station[3].%X2 )
      S_SR(operand := #SB1_1R2PutToolDone, r1 := wire#w1)
   END_RUNG
   RUNG wire#powerrail
      I_Contact( "HMI_CMD_Zone100".StationsSum.ModeChangeTools )
   END_RUNG wire#w1
   // the same network as SCL:
   IF "STATUS_1R2".Interlocks.Station[3].%X2 THEN
       #SB1_1R2PutToolDone := TRUE;   // SR flip-flop
   END_IF;
   IF NOT "HMI_CMD_Zone100".StationsSum.ModeChangeTools THEN #SB1_1R2PutToolDone := FALSE; END_IF;
END_REGION

REGION Network 24: Robot RO01 - switch tool done
   RUNG wire#powerrail
      Contact( "STATUS_1R2".Interlocks.Station[5].%X2 )
      wire#w1
      S_SR(operand := #SB1_1R1ToolSwitchDone, r1 := wire#w2)
   END_RUNG
   RUNG wire#powerrail
      Contact( "STATUS_1R2".Interlocks.Station[5].%X4 )
   END_RUNG wire#w1
   RUNG wire#powerrail
      I_Contact( "HMI_CMD_Zone100".StationsSum.ModeChangeTools )
   END_RUNG wire#w2
   // the same network as SCL:
   IF "STATUS_1R2".Interlocks.Station[5].%X2 OR "STATUS_1R2".Interlocks.Station[5].%X4 THEN
       #SB1_1R1ToolSwitchDone := TRUE;   // SR flip-flop
   END_IF;
   IF NOT "HMI_CMD_Zone100".StationsSum.ModeChangeTools THEN #SB1_1R1ToolSwitchDone := FALSE; END_IF;
END_REGION

REGION Network 25: Robot RO01 - request take parts from station 120
   RUNG wire#powerrail
      Contact( "STATUS_Zone100".Station1R2_Mode.Main.AutoRun )
      Contact( "STATUS_120".MatCard[1, 1].Occupied )
      Contact( #TB1GripperFree )
      Coil( #TB1Take120 )
   END_RUNG
   // the same network as SCL:
   #TB1Take120 := "STATUS_Zone100".Station1R2_Mode.Main.AutoRun AND "STATUS_120".MatCard[1, 1].Occupied AND #TB1GripperFree;
END_REGION

REGION Network 26: Robot RO01 - put position in 140 evaluation
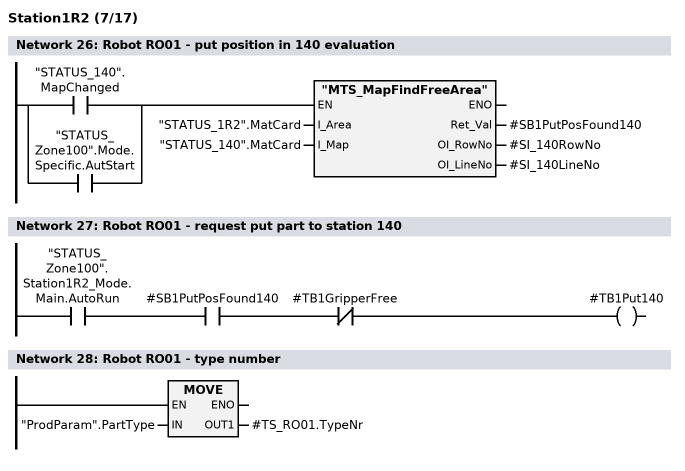
   RUNG wire#powerrail
      Contact( "STATUS_140".MapChanged )
      wire#w1
      "MTS_MapFindFreeArea"(I_Area := "STATUS_1R2".MatCard, I_Map := "STATUS_140".MatCard, Ret_Val => #SB1PutPosFound140, OI_RowNo => #SI_140RowNo, OI_LineNo => #SI_140LineNo)
   END_RUNG
   RUNG wire#powerrail
      Contact( "STATUS_Zone100".Mode.Specific.AutStart )
   END_RUNG wire#w1
   // the same network as SCL:
   IF "STATUS_140".MapChanged OR "STATUS_Zone100".Mode.Specific.AutStart THEN
       #SB1PutPosFound140 := "MTS_MapFindFreeArea"(I_Area := "STATUS_1R2".MatCard,
                               I_Map := "STATUS_140".MatCard,
                               OI_RowNo => #SI_140RowNo,
                               OI_LineNo => #SI_140LineNo);
   END_IF;
END_REGION

REGION Network 27: Robot RO01 - request put part to station 140
   RUNG wire#powerrail
      Contact( "STATUS_Zone100".Station1R2_Mode.Main.AutoRun )
      Contact( #SB1PutPosFound140 )
      I_Contact( #TB1GripperFree )
      Coil( #TB1Put140 )
   END_RUNG
   // the same network as SCL:
   #TB1Put140 := "STATUS_Zone100".Station1R2_Mode.Main.AutoRun AND #SB1PutPosFound140 AND NOT #TB1GripperFree;
END_REGION

REGION Network 28: Robot RO01 - type number
   RUNG wire#powerrail
      Move(in := "ProdParam".PartType, out1 => #TS_RO01.TypeNr)
   END_RUNG
   // the same network as SCL:
   #TS_RO01.TypeNr := "ProdParam".PartType;
END_REGION

REGION Network 29: Robot RO01 - start job
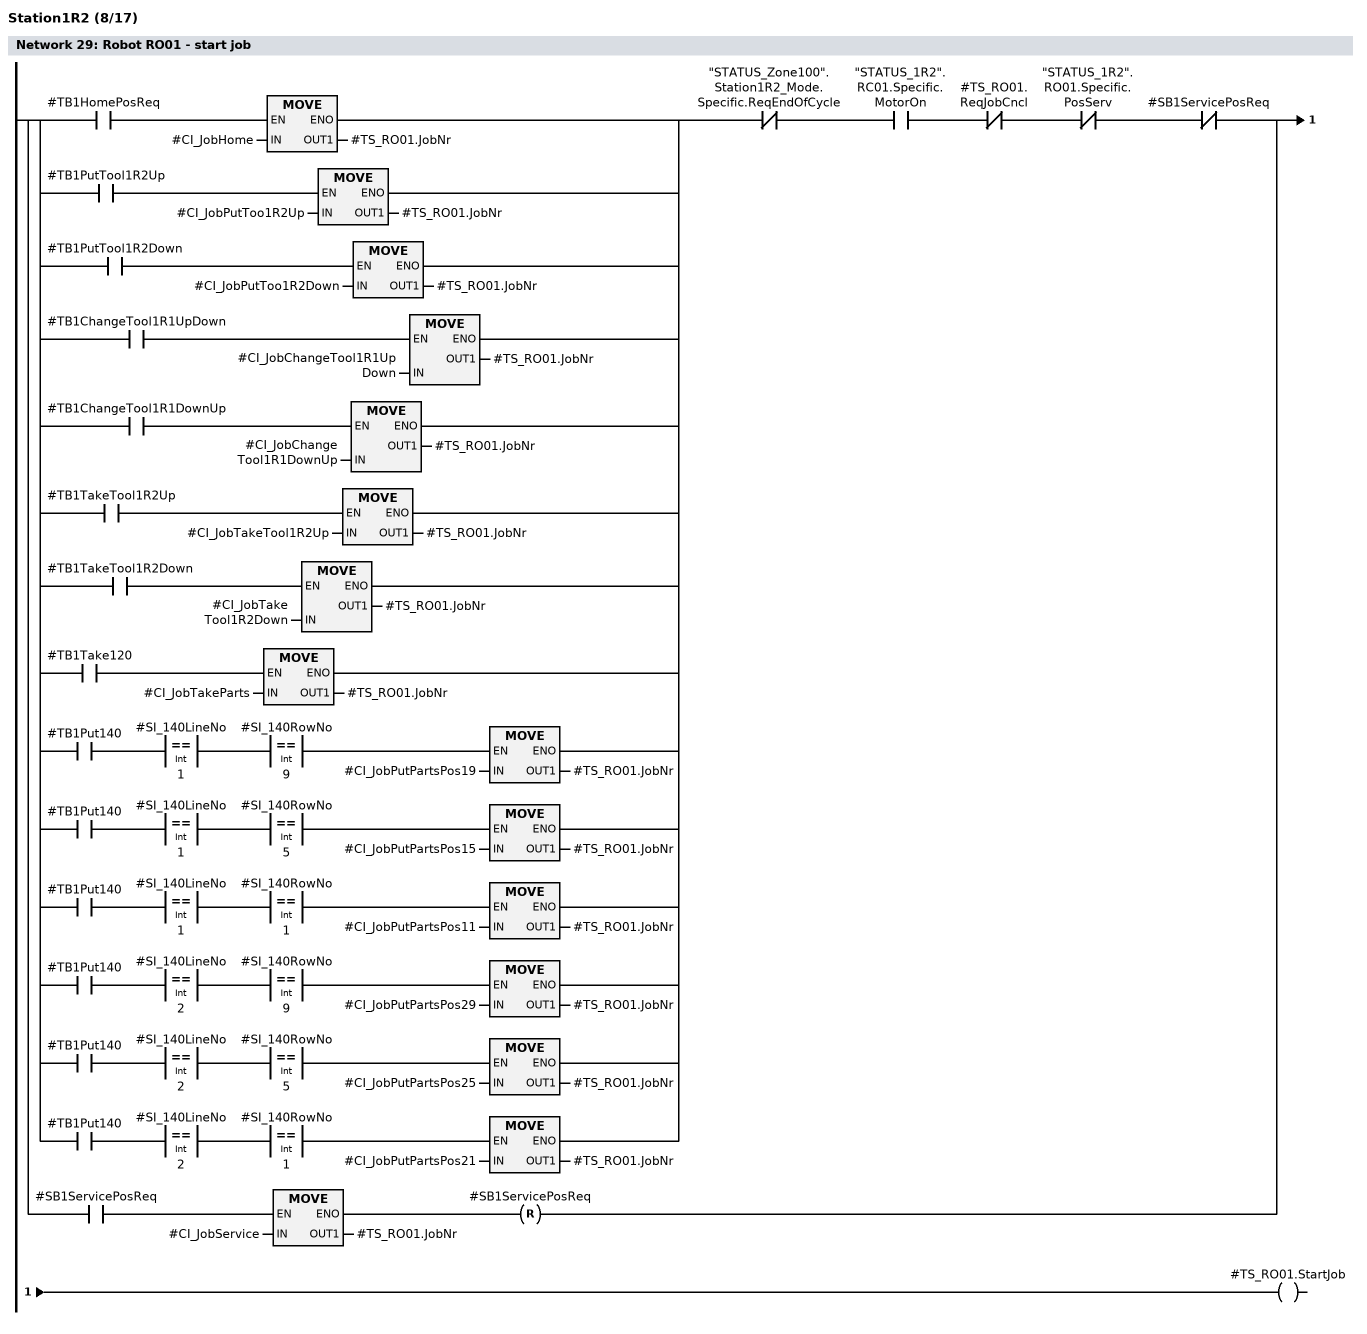
   RUNG wire#powerrail
      Contact( #TB1HomePosReq )
      Move(in := #CI_JobHome, out1 => #TS_RO01.JobNr)
      wire#w1
      I_Contact( "STATUS_Zone100".Station1R2_Mode.Specific.ReqEndOfCycle )
      Contact( "STATUS_1R2".RC01.Specific.MotorOn )
      I_Contact( #TS_RO01.ReqJobCncl )
      I_Contact( "STATUS_1R2".RO01.Specific.PosServ )
      I_Contact( #SB1ServicePosReq )
      wire#w2
      Coil( #TS_RO01.StartJob )
   END_RUNG
   RUNG wire#powerrail
      Contact( #TB1PutTool1R2Up )
      Move(in := #CI_JobPutToo1R2Up, out1 => #TS_RO01.JobNr)
   END_RUNG wire#w1
   RUNG wire#powerrail
      Contact( #TB1PutTool1R2Down )
      Move(in := #CI_JobPutToo1R2Down, out1 => #TS_RO01.JobNr)
   END_RUNG wire#w1
   RUNG wire#powerrail
      Contact( #TB1ChangeTool1R1UpDown )
      Move(in := #CI_JobChangeTool1R1UpDown, out1 => #TS_RO01.JobNr)
   END_RUNG wire#w1
   RUNG wire#powerrail
      Contact( #TB1ChangeTool1R1DownUp )
      Move(in := #CI_JobChangeTool1R1DownUp, out1 => #TS_RO01.JobNr)
   END_RUNG wire#w1
   RUNG wire#powerrail
      Contact( #TB1TakeTool1R2Up )
      Move(in := #CI_JobTakeTool1R2Up, out1 => #TS_RO01.JobNr)
   END_RUNG wire#w1
   RUNG wire#powerrail
      Contact( #TB1TakeTool1R2Down )
      Move(in := #CI_JobTakeTool1R2Down, out1 => #TS_RO01.JobNr)
   END_RUNG wire#w1
   RUNG wire#powerrail
      Contact( #TB1Take120 )
      Move(in := #CI_JobTakeParts, out1 => #TS_RO01.JobNr)
   END_RUNG wire#w1
   RUNG wire#powerrail
      Contact( #TB1Put140 )
      { S7_Templates := "SrcType := Int" } EQ_Contact(in1 := #SI_140LineNo, in2 := 1)
      { S7_Templates := "SrcType := Int" } EQ_Contact(in1 := #SI_140RowNo, in2 := 9)
      Move(in := #CI_JobPutPartsPos19, out1 => #TS_RO01.JobNr)
   END_RUNG wire#w1
   RUNG wire#powerrail
      Contact( #TB1Put140 )
      { S7_Templates := "SrcType := Int" } EQ_Contact(in1 := #SI_140LineNo, in2 := 1)
      { S7_Templates := "SrcType := Int" } EQ_Contact(in1 := #SI_140RowNo, in2 := 5)
      Move(in := #CI_JobPutPartsPos15, out1 => #TS_RO01.JobNr)
   END_RUNG wire#w1
   RUNG wire#powerrail
      Contact( #TB1Put140 )
      { S7_Templates := "SrcType := Int" } EQ_Contact(in1 := #SI_140LineNo, in2 := 1)
      { S7_Templates := "SrcType := Int" } EQ_Contact(in1 := #SI_140RowNo, in2 := 1)
      Move(in := #CI_JobPutPartsPos11, out1 => #TS_RO01.JobNr)
   END_RUNG wire#w1
   RUNG wire#powerrail
      Contact( #TB1Put140 )
      { S7_Templates := "SrcType := Int" } EQ_Contact(in1 := #SI_140LineNo, in2 := 2)
      { S7_Templates := "SrcType := Int" } EQ_Contact(in1 := #SI_140RowNo, in2 := 9)
      Move(in := #CI_JobPutPartsPos29, out1 => #TS_RO01.JobNr)
   END_RUNG wire#w1
   RUNG wire#powerrail
      Contact( #TB1Put140 )
      { S7_Templates := "SrcType := Int" } EQ_Contact(in1 := #SI_140LineNo, in2 := 2)
      { S7_Templates := "SrcType := Int" } EQ_Contact(in1 := #SI_140RowNo, in2 := 5)
      Move(in := #CI_JobPutPartsPos25, out1 => #TS_RO01.JobNr)
   END_RUNG wire#w1
   RUNG wire#powerrail
      Contact( #TB1Put140 )
      { S7_Templates := "SrcType := Int" } EQ_Contact(in1 := #SI_140LineNo, in2 := 2)
      { S7_Templates := "SrcType := Int" } EQ_Contact(in1 := #SI_140RowNo, in2 := 1)
      Move(in := #CI_JobPutPartsPos21, out1 => #TS_RO01.JobNr)
   END_RUNG wire#w1
   RUNG wire#powerrail
      Contact( #SB1ServicePosReq )
      Move(in := #CI_JobService, out1 => #TS_RO01.JobNr)
      R_Coil( #SB1ServicePosReq )
   END_RUNG wire#w2
   // the same network as SCL:
   IF #TB1HomePosReq THEN #TS_RO01.JobNr := #CI_JobHome; END_IF;
   IF #TB1PutTool1R2Up THEN #TS_RO01.JobNr := #CI_JobPutToo1R2Up; END_IF;
   IF #TB1PutTool1R2Down THEN #TS_RO01.JobNr := #CI_JobPutToo1R2Down; END_IF;
   IF #TB1ChangeTool1R1UpDown THEN #TS_RO01.JobNr := #CI_JobChangeTool1R1UpDown; END_IF;
   IF #TB1ChangeTool1R1DownUp THEN #TS_RO01.JobNr := #CI_JobChangeTool1R1DownUp; END_IF;
   IF #TB1TakeTool1R2Up THEN #TS_RO01.JobNr := #CI_JobTakeTool1R2Up; END_IF;
   IF #TB1TakeTool1R2Down THEN #TS_RO01.JobNr := #CI_JobTakeTool1R2Down; END_IF;
   IF #TB1Take120 THEN #TS_RO01.JobNr := #CI_JobTakeParts; END_IF;
   #_w1 := #TB1Put140 AND (#SI_140LineNo = 1) AND (#SI_140RowNo = 9);
   IF #_w1 THEN #TS_RO01.JobNr := #CI_JobPutPartsPos19; END_IF;
   #_w2 := #TB1Put140 AND (#SI_140LineNo = 1) AND (#SI_140RowNo = 5);
   IF #_w2 THEN #TS_RO01.JobNr := #CI_JobPutPartsPos15; END_IF;
   #_w3 := #TB1Put140 AND (#SI_140LineNo = 1) AND (#SI_140RowNo = 1);
   IF #_w3 THEN #TS_RO01.JobNr := #CI_JobPutPartsPos11; END_IF;
   #_w4 := #TB1Put140 AND (#SI_140LineNo = 2) AND (#SI_140RowNo = 9);
   IF #_w4 THEN #TS_RO01.JobNr := #CI_JobPutPartsPos29; END_IF;
   #_w5 := #TB1Put140 AND (#SI_140LineNo = 2) AND (#SI_140RowNo = 5);
   IF #_w5 THEN #TS_RO01.JobNr := #CI_JobPutPartsPos25; END_IF;
   #_w6 := #TB1Put140 AND (#SI_140LineNo = 2) AND (#SI_140RowNo = 1);
   IF #_w6 THEN #TS_RO01.JobNr := #CI_JobPutPartsPos21; END_IF;
   IF #SB1ServicePosReq THEN #TS_RO01.JobNr := #CI_JobService; END_IF;
   #_w7 := #SB1ServicePosReq;
   #_w8 := (#TB1HomePosReq OR #TB1PutTool1R2Up OR #TB1PutTool1R2Down OR #TB1ChangeTool1R1UpDown OR #TB1ChangeTool1R1DownUp OR #TB1TakeTool1R2Up OR #TB1TakeTool1R2Down OR #TB1Take120 OR #_w1 OR #_w2 OR #_w3 OR #_w4 OR #_w5 OR #_w6) AND NOT "STATUS_Zone100".Station1R2_Mode.Specific.ReqEndOfCycle AND "STATUS_1R2".RC01.Specific.MotorOn AND NOT #TS_RO01.ReqJobCncl AND NOT "STATUS_1R2".RO01.Specific.PosServ AND NOT #SB1ServicePosReq;
   IF #_w7 THEN #SB1ServicePosReq := FALSE; END_IF;
   #TS_RO01.StartJob := #_w8 OR #_w7;
END_REGION

REGION Network 30: *************** Interlocks ***************
END_REGION

REGION Network 31: Robot RO01 - interlocks - 120
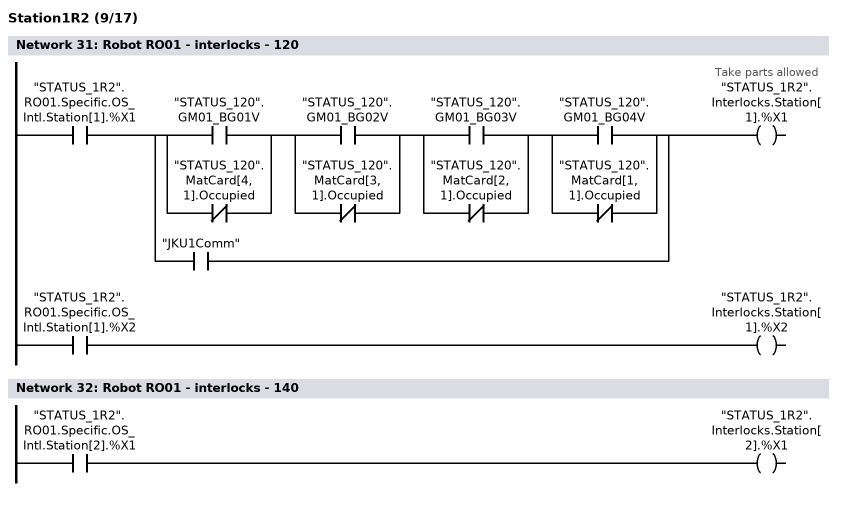
   RUNG wire#powerrail
      Contact( "STATUS_1R2".RO01.Specific.OS_Intl.Station[1].%X1 )
      wire#w1
      Contact( "STATUS_120".GM01_BG01V )
      wire#w2
      Contact( "STATUS_120".GM01_BG02V )
      wire#w3
      Contact( "STATUS_120".GM01_BG03V )
      wire#w4
      Contact( "STATUS_120".GM01_BG04V )
      wire#w5
      Coil( "STATUS_1R2".Interlocks.Station[1].%X1 )   // Take parts allowed
   END_RUNG
   RUNG wire#w1
      I_Contact( "STATUS_120".MatCard[4, 1].Occupied )
   END_RUNG wire#w2
   RUNG wire#w2
      I_Contact( "STATUS_120".MatCard[3, 1].Occupied )
   END_RUNG wire#w3
   RUNG wire#w3
      I_Contact( "STATUS_120".MatCard[2, 1].Occupied )
   END_RUNG wire#w4
   RUNG wire#w4
      I_Contact( "STATUS_120".MatCard[1, 1].Occupied )
   END_RUNG wire#w5
   RUNG wire#w1
      Contact( "JKU1Comm" )
   END_RUNG wire#w5
   RUNG wire#powerrail
      Contact( "STATUS_1R2".RO01.Specific.OS_Intl.Station[1].%X2 )
      Coil( "STATUS_1R2".Interlocks.Station[1].%X2 )
   END_RUNG
   // the same network as SCL:
   "STATUS_1R2".Interlocks.Station[1].%X1 := "STATUS_1R2".RO01.Specific.OS_Intl.Station[1].%X1 AND ((("STATUS_120".GM01_BG01V OR NOT "STATUS_120".MatCard[4, 1].Occupied) AND ("STATUS_120".GM01_BG02V OR NOT "STATUS_120".MatCard[3, 1].Occupied) AND ("STATUS_120".GM01_BG03V OR NOT "STATUS_120".MatCard[2, 1].Occupied) AND ("STATUS_120".GM01_BG04V OR NOT "STATUS_120".MatCard[1, 1].Occupied)) OR "JKU1Comm");   // Take parts allowed
   "STATUS_1R2".Interlocks.Station[1].%X2 := "STATUS_1R2".RO01.Specific.OS_Intl.Station[1].%X2;
END_REGION

REGION Network 32: Robot RO01 - interlocks - 140
   RUNG wire#powerrail
      Contact( "STATUS_1R2".RO01.Specific.OS_Intl.Station[2].%X1 )
      Coil( "STATUS_1R2".Interlocks.Station[2].%X1 )
   END_RUNG
   // the same network as SCL:
   "STATUS_1R2".Interlocks.Station[2].%X1 := "STATUS_1R2".RO01.Specific.OS_Intl.Station[2].%X1;
END_REGION

REGION Network 33: Robot RO01 - interlocks - CL01
   // "JSA0Comm" - add signal gripper on robot
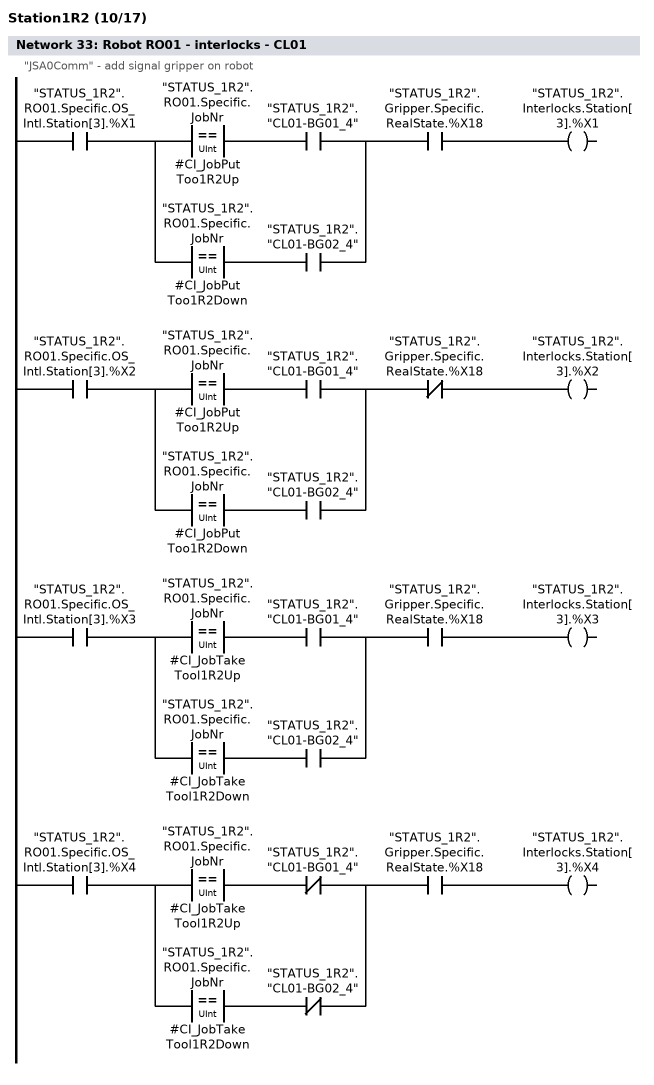
   RUNG wire#powerrail
      Contact( "STATUS_1R2".RO01.Specific.OS_Intl.Station[3].%X1 )
      wire#w1
      { S7_Templates := "SrcType := UInt" } EQ_Contact(in1 := "STATUS_1R2".RO01.Specific.JobNr, in2 := #CI_JobPutToo1R2Up)
      Contact( "STATUS_1R2"."CL01-BG01_4" )
      wire#w2
      Contact( "STATUS_1R2".Gripper.Specific.RealState.%X18 )
      Coil( "STATUS_1R2".Interlocks.Station[3].%X1 )
   END_RUNG
   RUNG wire#w1
      { S7_Templates := "SrcType := UInt" } EQ_Contact(in1 := "STATUS_1R2".RO01.Specific.JobNr, in2 := #CI_JobPutToo1R2Down)
      Contact( "STATUS_1R2"."CL01-BG02_4" )
   END_RUNG wire#w2
   RUNG wire#powerrail
      Contact( "STATUS_1R2".RO01.Specific.OS_Intl.Station[3].%X2 )
      wire#w3
      { S7_Templates := "SrcType := UInt" } EQ_Contact(in1 := "STATUS_1R2".RO01.Specific.JobNr, in2 := #CI_JobPutToo1R2Up)
      Contact( "STATUS_1R2"."CL01-BG01_4" )
      wire#w4
      I_Contact( "STATUS_1R2".Gripper.Specific.RealState.%X18 )
      Coil( "STATUS_1R2".Interlocks.Station[3].%X2 )
   END_RUNG
   RUNG wire#w3
      { S7_Templates := "SrcType := UInt" } EQ_Contact(in1 := "STATUS_1R2".RO01.Specific.JobNr, in2 := #CI_JobPutToo1R2Down)
      Contact( "STATUS_1R2"."CL01-BG02_4" )
   END_RUNG wire#w4
   RUNG wire#powerrail
      Contact( "STATUS_1R2".RO01.Specific.OS_Intl.Station[3].%X3 )
      wire#w5
      { S7_Templates := "SrcType := UInt" } EQ_Contact(in1 := "STATUS_1R2".RO01.Specific.JobNr, in2 := #CI_JobTakeTool1R2Up)
      Contact( "STATUS_1R2"."CL01-BG01_4" )
      wire#w6
      Contact( "STATUS_1R2".Gripper.Specific.RealState.%X18 )
      Coil( "STATUS_1R2".Interlocks.Station[3].%X3 )
   END_RUNG
   RUNG wire#w5
      { S7_Templates := "SrcType := UInt" } EQ_Contact(in1 := "STATUS_1R2".RO01.Specific.JobNr, in2 := #CI_JobTakeTool1R2Down)
      Contact( "STATUS_1R2"."CL01-BG02_4" )
   END_RUNG wire#w6
   RUNG wire#powerrail
      Contact( "STATUS_1R2".RO01.Specific.OS_Intl.Station[3].%X4 )
      wire#w7
      { S7_Templates := "SrcType := UInt" } EQ_Contact(in1 := "STATUS_1R2".RO01.Specific.JobNr, in2 := #CI_JobTakeTool1R2Up)
      I_Contact( "STATUS_1R2"."CL01-BG01_4" )
      wire#w8
      Contact( "STATUS_1R2".Gripper.Specific.RealState.%X18 )
      Coil( "STATUS_1R2".Interlocks.Station[3].%X4 )
   END_RUNG
   RUNG wire#w7
      { S7_Templates := "SrcType := UInt" } EQ_Contact(in1 := "STATUS_1R2".RO01.Specific.JobNr, in2 := #CI_JobTakeTool1R2Down)
      I_Contact( "STATUS_1R2"."CL01-BG02_4" )
   END_RUNG wire#w8
   // the same network as SCL:
   "STATUS_1R2".Interlocks.Station[3].%X1 := "STATUS_1R2".RO01.Specific.OS_Intl.Station[3].%X1 AND ((("STATUS_1R2".RO01.Specific.JobNr = #CI_JobPutToo1R2Up) AND "STATUS_1R2"."CL01-BG01_4") OR (("STATUS_1R2".RO01.Specific.JobNr = #CI_JobPutToo1R2Down) AND "STATUS_1R2"."CL01-BG02_4")) AND "STATUS_1R2".Gripper.Specific.RealState.%X18;
   "STATUS_1R2".Interlocks.Station[3].%X2 := "STATUS_1R2".RO01.Specific.OS_Intl.Station[3].%X2 AND ((("STATUS_1R2".RO01.Specific.JobNr = #CI_JobPutToo1R2Up) AND "STATUS_1R2"."CL01-BG01_4") OR (("STATUS_1R2".RO01.Specific.JobNr = #CI_JobPutToo1R2Down) AND "STATUS_1R2"."CL01-BG02_4")) AND NOT "STATUS_1R2".Gripper.Specific.RealState.%X18;
   "STATUS_1R2".Interlocks.Station[3].%X3 := "STATUS_1R2".RO01.Specific.OS_Intl.Station[3].%X3 AND ((("STATUS_1R2".RO01.Specific.JobNr = #CI_JobTakeTool1R2Up) AND "STATUS_1R2"."CL01-BG01_4") OR (("STATUS_1R2".RO01.Specific.JobNr = #CI_JobTakeTool1R2Down) AND "STATUS_1R2"."CL01-BG02_4")) AND "STATUS_1R2".Gripper.Specific.RealState.%X18;
   "STATUS_1R2".Interlocks.Station[3].%X4 := "STATUS_1R2".RO01.Specific.OS_Intl.Station[3].%X4 AND ((("STATUS_1R2".RO01.Specific.JobNr = #CI_JobTakeTool1R2Up) AND NOT "STATUS_1R2"."CL01-BG01_4") OR (("STATUS_1R2".RO01.Specific.JobNr = #CI_JobTakeTool1R2Down) AND NOT "STATUS_1R2"."CL01-BG02_4")) AND "STATUS_1R2".Gripper.Specific.RealState.%X18;
END_REGION

REGION Network 34: Robot RO01 - interlocks - 1R1+CL01
   // "JSA0Comm" - add signal gripper on robot
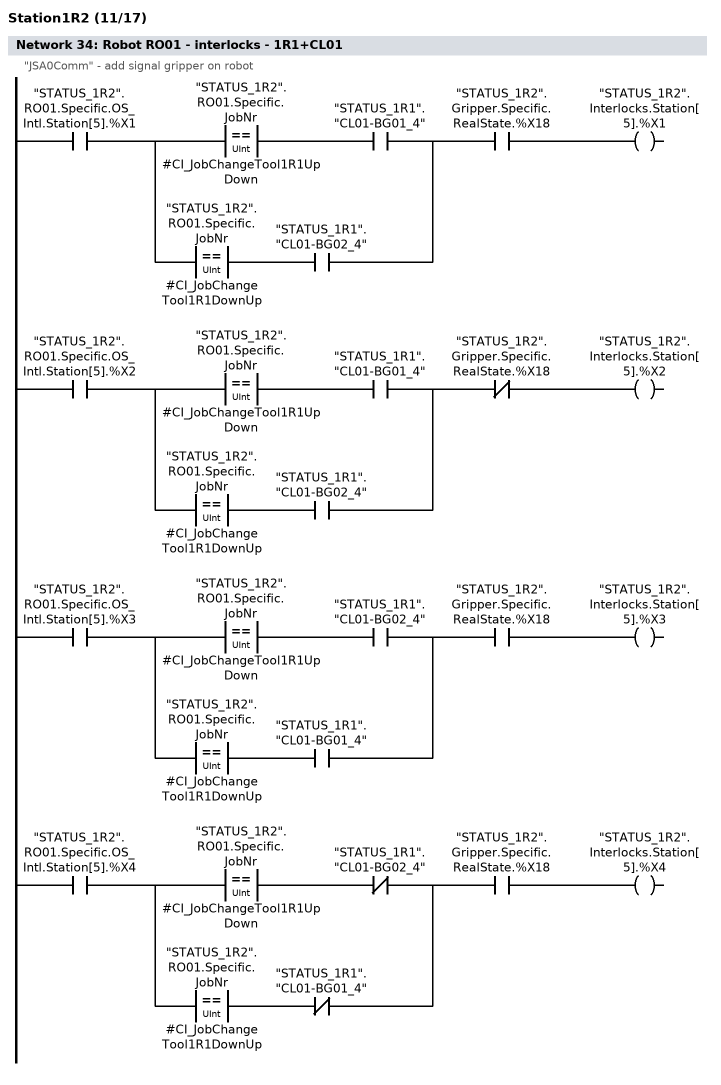
   RUNG wire#powerrail
      Contact( "STATUS_1R2".RO01.Specific.OS_Intl.Station[5].%X1 )
      wire#w1
      { S7_Templates := "SrcType := UInt" } EQ_Contact(in1 := "STATUS_1R2".RO01.Specific.JobNr, in2 := #CI_JobChangeTool1R1UpDown)
      Contact( "STATUS_1R1"."CL01-BG01_4" )
      wire#w2
      Contact( "STATUS_1R2".Gripper.Specific.RealState.%X18 )
      Coil( "STATUS_1R2".Interlocks.Station[5].%X1 )
   END_RUNG
   RUNG wire#w1
      { S7_Templates := "SrcType := UInt" } EQ_Contact(in1 := "STATUS_1R2".RO01.Specific.JobNr, in2 := #CI_JobChangeTool1R1DownUp)
      Contact( "STATUS_1R1"."CL01-BG02_4" )
   END_RUNG wire#w2
   RUNG wire#powerrail
      Contact( "STATUS_1R2".RO01.Specific.OS_Intl.Station[5].%X2 )
      wire#w3
      { S7_Templates := "SrcType := UInt" } EQ_Contact(in1 := "STATUS_1R2".RO01.Specific.JobNr, in2 := #CI_JobChangeTool1R1UpDown)
      Contact( "STATUS_1R1"."CL01-BG01_4" )
      wire#w4
      I_Contact( "STATUS_1R2".Gripper.Specific.RealState.%X18 )
      Coil( "STATUS_1R2".Interlocks.Station[5].%X2 )
   END_RUNG
   RUNG wire#w3
      { S7_Templates := "SrcType := UInt" } EQ_Contact(in1 := "STATUS_1R2".RO01.Specific.JobNr, in2 := #CI_JobChangeTool1R1DownUp)
      Contact( "STATUS_1R1"."CL01-BG02_4" )
   END_RUNG wire#w4
   RUNG wire#powerrail
      Contact( "STATUS_1R2".RO01.Specific.OS_Intl.Station[5].%X3 )
      wire#w5
      { S7_Templates := "SrcType := UInt" } EQ_Contact(in1 := "STATUS_1R2".RO01.Specific.JobNr, in2 := #CI_JobChangeTool1R1UpDown)
      Contact( "STATUS_1R1"."CL01-BG02_4" )
      wire#w6
      Contact( "STATUS_1R2".Gripper.Specific.RealState.%X18 )
      Coil( "STATUS_1R2".Interlocks.Station[5].%X3 )
   END_RUNG
   RUNG wire#w5
      { S7_Templates := "SrcType := UInt" } EQ_Contact(in1 := "STATUS_1R2".RO01.Specific.JobNr, in2 := #CI_JobChangeTool1R1DownUp)
      Contact( "STATUS_1R1"."CL01-BG01_4" )
   END_RUNG wire#w6
   RUNG wire#powerrail
      Contact( "STATUS_1R2".RO01.Specific.OS_Intl.Station[5].%X4 )
      wire#w7
      { S7_Templates := "SrcType := UInt" } EQ_Contact(in1 := "STATUS_1R2".RO01.Specific.JobNr, in2 := #CI_JobChangeTool1R1UpDown)
      I_Contact( "STATUS_1R1"."CL01-BG02_4" )
      wire#w8
      Contact( "STATUS_1R2".Gripper.Specific.RealState.%X18 )
      Coil( "STATUS_1R2".Interlocks.Station[5].%X4 )
   END_RUNG
   RUNG wire#w7
      { S7_Templates := "SrcType := UInt" } EQ_Contact(in1 := "STATUS_1R2".RO01.Specific.JobNr, in2 := #CI_JobChangeTool1R1DownUp)
      I_Contact( "STATUS_1R1"."CL01-BG01_4" )
   END_RUNG wire#w8
   // the same network as SCL:
   "STATUS_1R2".Interlocks.Station[5].%X1 := "STATUS_1R2".RO01.Specific.OS_Intl.Station[5].%X1 AND ((("STATUS_1R2".RO01.Specific.JobNr = #CI_JobChangeTool1R1UpDown) AND "STATUS_1R1"."CL01-BG01_4") OR (("STATUS_1R2".RO01.Specific.JobNr = #CI_JobChangeTool1R1DownUp) AND "STATUS_1R1"."CL01-BG02_4")) AND "STATUS_1R2".Gripper.Specific.RealState.%X18;
   "STATUS_1R2".Interlocks.Station[5].%X2 := "STATUS_1R2".RO01.Specific.OS_Intl.Station[5].%X2 AND ((("STATUS_1R2".RO01.Specific.JobNr = #CI_JobChangeTool1R1UpDown) AND "STATUS_1R1"."CL01-BG01_4") OR (("STATUS_1R2".RO01.Specific.JobNr = #CI_JobChangeTool1R1DownUp) AND "STATUS_1R1"."CL01-BG02_4")) AND NOT "STATUS_1R2".Gripper.Specific.RealState.%X18;
   "STATUS_1R2".Interlocks.Station[5].%X3 := "STATUS_1R2".RO01.Specific.OS_Intl.Station[5].%X3 AND ((("STATUS_1R2".RO01.Specific.JobNr = #CI_JobChangeTool1R1UpDown) AND "STATUS_1R1"."CL01-BG02_4") OR (("STATUS_1R2".RO01.Specific.JobNr = #CI_JobChangeTool1R1DownUp) AND "STATUS_1R1"."CL01-BG01_4")) AND "STATUS_1R2".Gripper.Specific.RealState.%X18;
   "STATUS_1R2".Interlocks.Station[5].%X4 := "STATUS_1R2".RO01.Specific.OS_Intl.Station[5].%X4 AND ((("STATUS_1R2".RO01.Specific.JobNr = #CI_JobChangeTool1R1UpDown) AND NOT "STATUS_1R1"."CL01-BG02_4") OR (("STATUS_1R2".RO01.Specific.JobNr = #CI_JobChangeTool1R1DownUp) AND NOT "STATUS_1R1"."CL01-BG01_4")) AND "STATUS_1R2".Gripper.Specific.RealState.%X18;
END_REGION

REGION Network 35: Robot RO01 - interlocks - 1R1+CL02
   // "JSA0Comm" - add signal gripper on robot
   // "JSA0Comm" - add signal gripper on robot
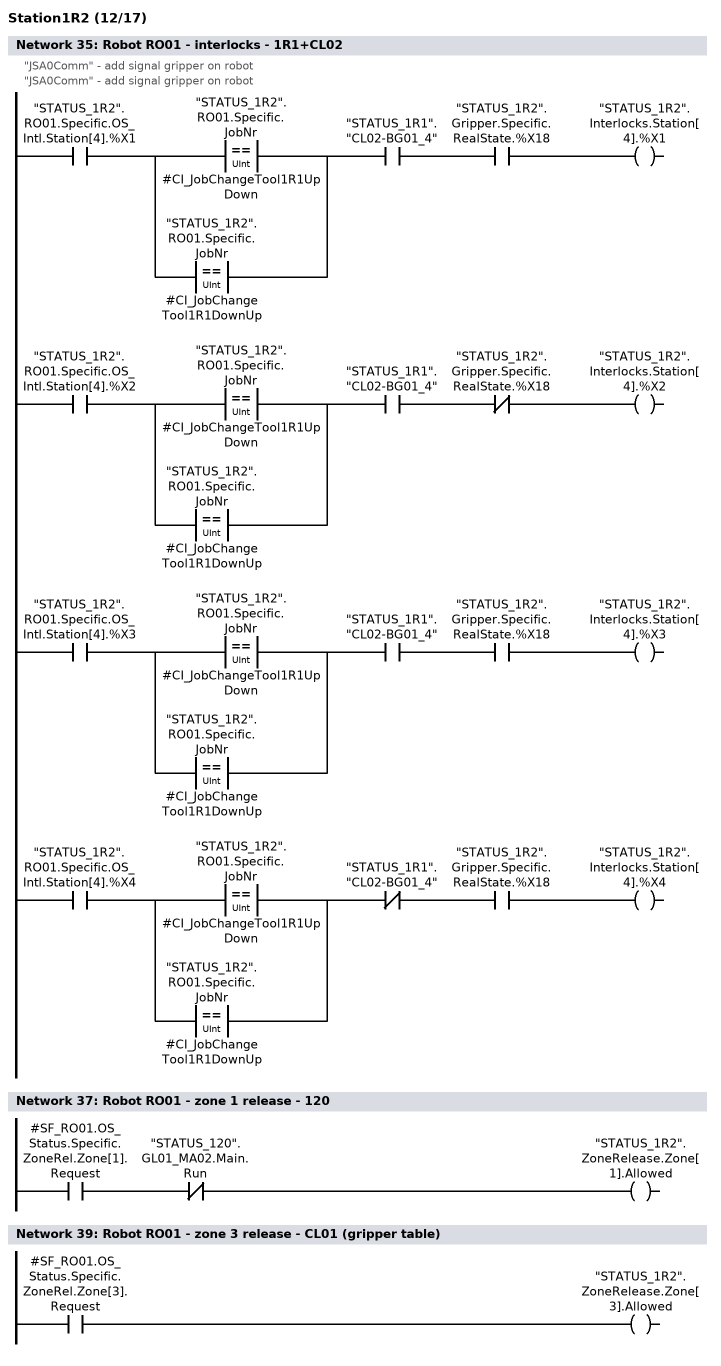
   RUNG wire#powerrail
      Contact( "STATUS_1R2".RO01.Specific.OS_Intl.Station[4].%X1 )
      wire#w1
      { S7_Templates := "SrcType := UInt" } EQ_Contact(in1 := "STATUS_1R2".RO01.Specific.JobNr, in2 := #CI_JobChangeTool1R1UpDown)
      wire#w2
      Contact( "STATUS_1R1"."CL02-BG01_4" )
      Contact( "STATUS_1R2".Gripper.Specific.RealState.%X18 )
      Coil( "STATUS_1R2".Interlocks.Station[4].%X1 )
   END_RUNG
   RUNG wire#w1
      { S7_Templates := "SrcType := UInt" } EQ_Contact(in1 := "STATUS_1R2".RO01.Specific.JobNr, in2 := #CI_JobChangeTool1R1DownUp)
   END_RUNG wire#w2
   RUNG wire#powerrail
      Contact( "STATUS_1R2".RO01.Specific.OS_Intl.Station[4].%X2 )
      wire#w3
      { S7_Templates := "SrcType := UInt" } EQ_Contact(in1 := "STATUS_1R2".RO01.Specific.JobNr, in2 := #CI_JobChangeTool1R1UpDown)
      wire#w4
      Contact( "STATUS_1R1"."CL02-BG01_4" )
      I_Contact( "STATUS_1R2".Gripper.Specific.RealState.%X18 )
      Coil( "STATUS_1R2".Interlocks.Station[4].%X2 )
   END_RUNG
   RUNG wire#w3
      { S7_Templates := "SrcType := UInt" } EQ_Contact(in1 := "STATUS_1R2".RO01.Specific.JobNr, in2 := #CI_JobChangeTool1R1DownUp)
   END_RUNG wire#w4
   RUNG wire#powerrail
      Contact( "STATUS_1R2".RO01.Specific.OS_Intl.Station[4].%X3 )
      wire#w5
      { S7_Templates := "SrcType := UInt" } EQ_Contact(in1 := "STATUS_1R2".RO01.Specific.JobNr, in2 := #CI_JobChangeTool1R1UpDown)
      wire#w6
      Contact( "STATUS_1R1"."CL02-BG01_4" )
      Contact( "STATUS_1R2".Gripper.Specific.RealState.%X18 )
      Coil( "STATUS_1R2".Interlocks.Station[4].%X3 )
   END_RUNG
   RUNG wire#w5
      { S7_Templates := "SrcType := UInt" } EQ_Contact(in1 := "STATUS_1R2".RO01.Specific.JobNr, in2 := #CI_JobChangeTool1R1DownUp)
   END_RUNG wire#w6
   RUNG wire#powerrail
      Contact( "STATUS_1R2".RO01.Specific.OS_Intl.Station[4].%X4 )
      wire#w7
      { S7_Templates := "SrcType := UInt" } EQ_Contact(in1 := "STATUS_1R2".RO01.Specific.JobNr, in2 := #CI_JobChangeTool1R1UpDown)
      wire#w8
      I_Contact( "STATUS_1R1"."CL02-BG01_4" )
      Contact( "STATUS_1R2".Gripper.Specific.RealState.%X18 )
      Coil( "STATUS_1R2".Interlocks.Station[4].%X4 )
   END_RUNG
   RUNG wire#w7
      { S7_Templates := "SrcType := UInt" } EQ_Contact(in1 := "STATUS_1R2".RO01.Specific.JobNr, in2 := #CI_JobChangeTool1R1DownUp)
   END_RUNG wire#w8
   // the same network as SCL:
   "STATUS_1R2".Interlocks.Station[4].%X1 := "STATUS_1R2".RO01.Specific.OS_Intl.Station[4].%X1 AND (("STATUS_1R2".RO01.Specific.JobNr = #CI_JobChangeTool1R1UpDown) OR ("STATUS_1R2".RO01.Specific.JobNr = #CI_JobChangeTool1R1DownUp)) AND "STATUS_1R1"."CL02-BG01_4" AND "STATUS_1R2".Gripper.Specific.RealState.%X18;
   "STATUS_1R2".Interlocks.Station[4].%X2 := "STATUS_1R2".RO01.Specific.OS_Intl.Station[4].%X2 AND (("STATUS_1R2".RO01.Specific.JobNr = #CI_JobChangeTool1R1UpDown) OR ("STATUS_1R2".RO01.Specific.JobNr = #CI_JobChangeTool1R1DownUp)) AND "STATUS_1R1"."CL02-BG01_4" AND NOT "STATUS_1R2".Gripper.Specific.RealState.%X18;
   "STATUS_1R2".Interlocks.Station[4].%X3 := "STATUS_1R2".RO01.Specific.OS_Intl.Station[4].%X3 AND (("STATUS_1R2".RO01.Specific.JobNr = #CI_JobChangeTool1R1UpDown) OR ("STATUS_1R2".RO01.Specific.JobNr = #CI_JobChangeTool1R1DownUp)) AND "STATUS_1R1"."CL02-BG01_4" AND "STATUS_1R2".Gripper.Specific.RealState.%X18;
   "STATUS_1R2".Interlocks.Station[4].%X4 := "STATUS_1R2".RO01.Specific.OS_Intl.Station[4].%X4 AND (("STATUS_1R2".RO01.Specific.JobNr = #CI_JobChangeTool1R1UpDown) OR ("STATUS_1R2".RO01.Specific.JobNr = #CI_JobChangeTool1R1DownUp)) AND NOT "STATUS_1R1"."CL02-BG01_4" AND "STATUS_1R2".Gripper.Specific.RealState.%X18;
END_REGION

REGION Network 36: *************** Zone release *************
END_REGION

REGION Network 37: Robot RO01 - zone 1 release - 120
   RUNG wire#powerrail
      Contact( #SF_RO01.OS_Status.Specific.ZoneRel.Zone[1].Request )
      I_Contact( "STATUS_120".GL01_MA02.Main.Run )
      Coil( "STATUS_1R2".ZoneRelease.Zone[1].Allowed )
   END_RUNG
   // the same network as SCL:
   "STATUS_1R2".ZoneRelease.Zone[1].Allowed := #SF_RO01.OS_Status.Specific.ZoneRel.Zone[1].Request AND NOT "STATUS_120".GL01_MA02.Main.Run;
END_REGION

REGION Network 38: Robot RO01 - zone 2 release - 140 - evaluation in FB Station140
END_REGION

REGION Network 39: Robot RO01 - zone 3 release - CL01 (gripper table)
   RUNG wire#powerrail
      Contact( #SF_RO01.OS_Status.Specific.ZoneRel.Zone[3].Request )
      Coil( "STATUS_1R2".ZoneRelease.Zone[3].Allowed )
   END_RUNG
   // the same network as SCL:
   "STATUS_1R2".ZoneRelease.Zone[3].Allowed := #SF_RO01.OS_Status.Specific.ZoneRel.Zone[3].Request;
END_REGION

REGION Network 40: Robot RO01 - zone 4 release - 1R2+CL02 (gripper table) - evaluation in FB Station1R2
END_REGION

REGION Network 41: Robot RO01 - zone 5 release - 1R2+CL01 (gripper table)
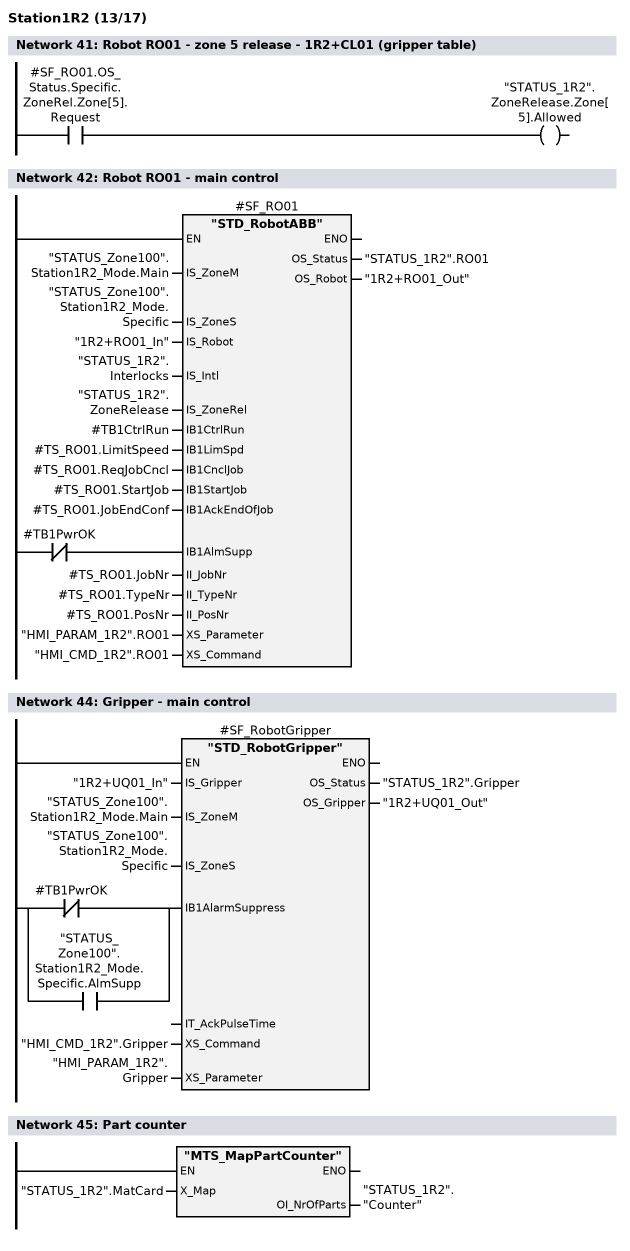
   RUNG wire#powerrail
      Contact( #SF_RO01.OS_Status.Specific.ZoneRel.Zone[5].Request )
      Coil( "STATUS_1R2".ZoneRelease.Zone[5].Allowed )
   END_RUNG
   // the same network as SCL:
   "STATUS_1R2".ZoneRelease.Zone[5].Allowed := #SF_RO01.OS_Status.Specific.ZoneRel.Zone[5].Request;
END_REGION

REGION Network 42: Robot RO01 - main control
   RUNG wire#powerrail
      #SF_RO01(IB1AlmSupp := wire#w1, IS_ZoneM := "STATUS_Zone100".Station1R2_Mode.Main, IS_ZoneS := "STATUS_Zone100".Station1R2_Mode.Specific, IS_Robot := "1R2+RO01_In", IS_Intl := "STATUS_1R2".Interlocks, IS_ZoneRel := "STATUS_1R2".ZoneRelease, IB1CtrlRun := #TB1CtrlRun, IB1LimSpd := #TS_RO01.LimitSpeed, IB1CnclJob := #TS_RO01.ReqJobCncl, IB1StartJob := #TS_RO01.StartJob, IB1AckEndOfJob := #TS_RO01.JobEndConf, II_JobNr := #TS_RO01.JobNr, II_TypeNr := #TS_RO01.TypeNr, II_PosNr := #TS_RO01.PosNr, XS_Parameter := "HMI_PARAM_1R2".RO01, XS_Command := "HMI_CMD_1R2".RO01, OS_Status => "STATUS_1R2".RO01, OS_Robot => "1R2+RO01_Out")
   END_RUNG
   RUNG wire#powerrail
      I_Contact( #TB1PwrOK )
   END_RUNG wire#w1
   // the same network as SCL:
   #SF_RO01(IS_ZoneM := "STATUS_Zone100".Station1R2_Mode.Main,   // "STD_RobotABB"
            IS_ZoneS := "STATUS_Zone100".Station1R2_Mode.Specific,
            IS_Robot := "1R2+RO01_In",
            IS_Intl := "STATUS_1R2".Interlocks,
            IS_ZoneRel := "STATUS_1R2".ZoneRelease,
            IB1CtrlRun := #TB1CtrlRun,
            IB1LimSpd := #TS_RO01.LimitSpeed,
            IB1CnclJob := #TS_RO01.ReqJobCncl,
            IB1StartJob := #TS_RO01.StartJob,
            IB1AckEndOfJob := #TS_RO01.JobEndConf,
            IB1AlmSupp := NOT #TB1PwrOK,
            II_JobNr := #TS_RO01.JobNr,
            II_TypeNr := #TS_RO01.TypeNr,
            II_PosNr := #TS_RO01.PosNr,
            XS_Parameter := "HMI_PARAM_1R2".RO01,
            XS_Command := "HMI_CMD_1R2".RO01,
            OS_Status => "STATUS_1R2".RO01,
            OS_Robot => "1R2+RO01_Out");
END_REGION

REGION Network 43: *************** Gripper ***************
END_REGION

REGION Network 44: Gripper - main control
   RUNG wire#powerrail
      #SF_RobotGripper(IB1AlarmSuppress := wire#w1, IS_Gripper := "1R2+UQ01_In", IS_ZoneM := "STATUS_Zone100".Station1R2_Mode.Main, IS_ZoneS := "STATUS_Zone100".Station1R2_Mode.Specific, IT_AckPulseTime :=, XS_Command := "HMI_CMD_1R2".Gripper, XS_Parameter := "HMI_PARAM_1R2".Gripper, OS_Status => "STATUS_1R2".Gripper, OS_Gripper => "1R2+UQ01_Out")
   END_RUNG
   RUNG wire#powerrail
      I_Contact( #TB1PwrOK )
   END_RUNG wire#w1
   RUNG wire#powerrail
      Contact( "STATUS_Zone100".Station1R2_Mode.Specific.AlmSupp )
   END_RUNG wire#w1
   // the same network as SCL:
   #SF_RobotGripper(IS_Gripper := "1R2+UQ01_In",   // "STD_RobotGripper"
                    IS_ZoneM := "STATUS_Zone100".Station1R2_Mode.Main,
                    IS_ZoneS := "STATUS_Zone100".Station1R2_Mode.Specific,
                    IB1AlarmSuppress := NOT #TB1PwrOK OR "STATUS_Zone100".Station1R2_Mode.Specific.AlmSupp,
                    XS_Command := "HMI_CMD_1R2".Gripper,
                    XS_Parameter := "HMI_PARAM_1R2".Gripper,
                    OS_Status => "STATUS_1R2".Gripper,
                    OS_Gripper => "1R2+UQ01_Out");
END_REGION

REGION Network 45: Part counter
   RUNG wire#powerrail
      "MTS_MapPartCounter"(X_Map := "STATUS_1R2".MatCard, OI_NrOfParts => "STATUS_1R2"."Counter")
   END_RUNG
   // the same network as SCL:
   "MTS_MapPartCounter"(X_Map := "STATUS_1R2".MatCard, OI_NrOfParts => "STATUS_1R2"."Counter");
END_REGION

REGION Network 46: *************** Material flow ***************
END_REGION

REGION Network 47: Clear positions and map - commands
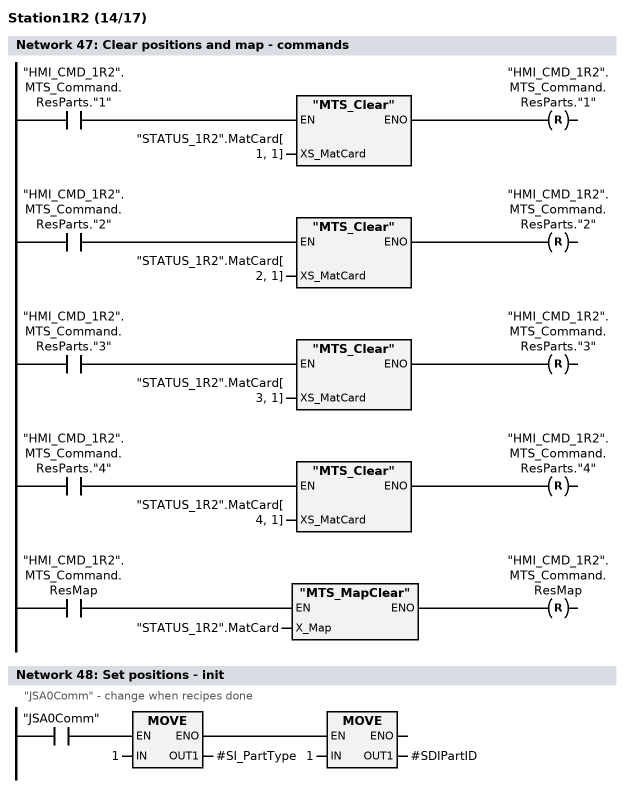
   RUNG wire#powerrail
      Contact( "HMI_CMD_1R2".MTS_Command.ResParts."1" )
      "MTS_Clear"(XS_MatCard := "STATUS_1R2".MatCard[1, 1])
      R_Coil( "HMI_CMD_1R2".MTS_Command.ResParts."1" )
   END_RUNG
   RUNG wire#powerrail
      Contact( "HMI_CMD_1R2".MTS_Command.ResParts."2" )
      "MTS_Clear"(XS_MatCard := "STATUS_1R2".MatCard[2, 1])
      R_Coil( "HMI_CMD_1R2".MTS_Command.ResParts."2" )
   END_RUNG
   RUNG wire#powerrail
      Contact( "HMI_CMD_1R2".MTS_Command.ResParts."3" )
      "MTS_Clear"(XS_MatCard := "STATUS_1R2".MatCard[3, 1])
      R_Coil( "HMI_CMD_1R2".MTS_Command.ResParts."3" )
   END_RUNG
   RUNG wire#powerrail
      Contact( "HMI_CMD_1R2".MTS_Command.ResParts."4" )
      "MTS_Clear"(XS_MatCard := "STATUS_1R2".MatCard[4, 1])
      R_Coil( "HMI_CMD_1R2".MTS_Command.ResParts."4" )
   END_RUNG
   RUNG wire#powerrail
      Contact( "HMI_CMD_1R2".MTS_Command.ResMap )
      "MTS_MapClear"(X_Map := "STATUS_1R2".MatCard)
      R_Coil( "HMI_CMD_1R2".MTS_Command.ResMap )
   END_RUNG
   // the same network as SCL:
   "MTS_Clear"(EN := "HMI_CMD_1R2".MTS_Command.ResParts."1",
               XS_MatCard := "STATUS_1R2".MatCard[1, 1],
               ENO => #_w1);
   IF #_w1 THEN "HMI_CMD_1R2".MTS_Command.ResParts."1" := FALSE; END_IF;
   "MTS_Clear"(EN := "HMI_CMD_1R2".MTS_Command.ResParts."2",
               XS_MatCard := "STATUS_1R2".MatCard[2, 1],
               ENO => #_w2);
   IF #_w2 THEN "HMI_CMD_1R2".MTS_Command.ResParts."2" := FALSE; END_IF;
   "MTS_Clear"(EN := "HMI_CMD_1R2".MTS_Command.ResParts."3",
               XS_MatCard := "STATUS_1R2".MatCard[3, 1],
               ENO => #_w3);
   IF #_w3 THEN "HMI_CMD_1R2".MTS_Command.ResParts."3" := FALSE; END_IF;
   "MTS_Clear"(EN := "HMI_CMD_1R2".MTS_Command.ResParts."4",
               XS_MatCard := "STATUS_1R2".MatCard[4, 1],
               ENO => #_w4);
   IF #_w4 THEN "HMI_CMD_1R2".MTS_Command.ResParts."4" := FALSE; END_IF;
   "MTS_MapClear"(EN := "HMI_CMD_1R2".MTS_Command.ResMap, X_Map := "STATUS_1R2".MatCard, ENO => #_w5);
   IF #_w5 THEN "HMI_CMD_1R2".MTS_Command.ResMap := FALSE; END_IF;
END_REGION

REGION Network 48: Set positions - init
   // "JSA0Comm" - change when recipes done
   RUNG wire#powerrail
      Contact( "JSA0Comm" )
      Move(in := 1, out1 => #SI_PartType)
      Move(in := 1, out1 => #SDIPartID)
   END_RUNG
   // the same network as SCL:
   IF "JSA0Comm" THEN
       #SI_PartType := 1;
       #SDIPartID := 1;
   END_IF;
END_REGION

REGION Network 49: Set positions and map - commands
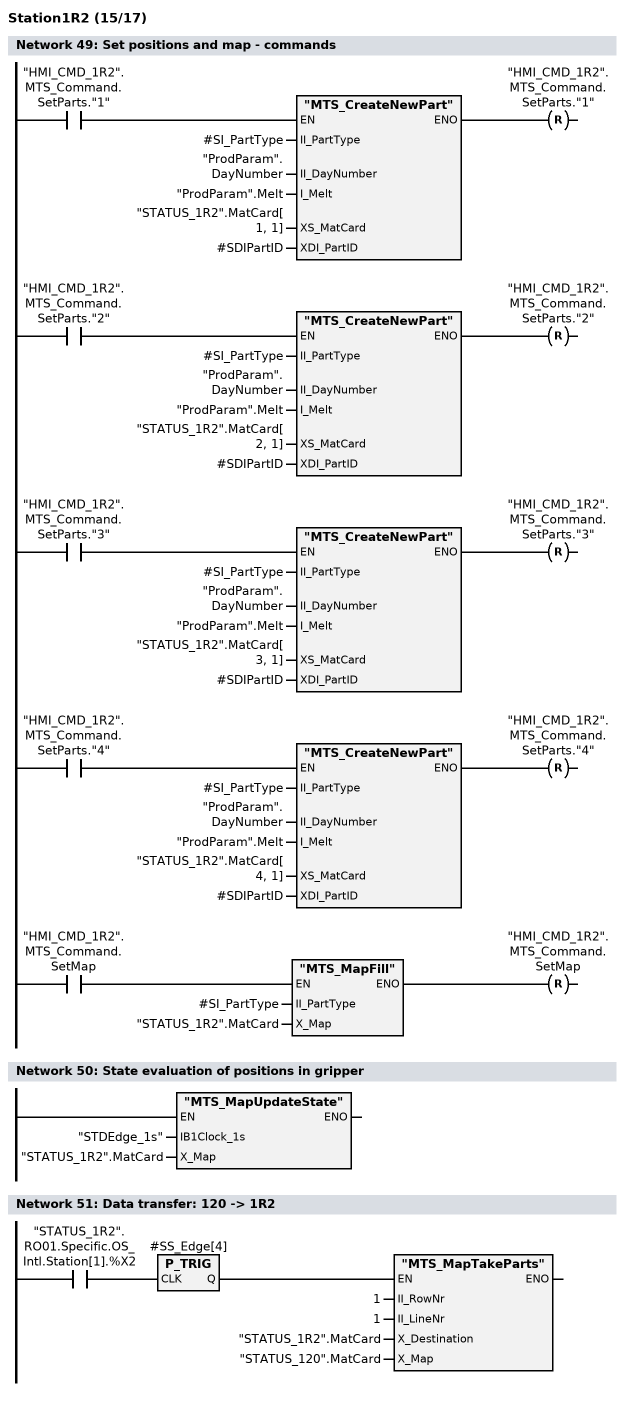
   RUNG wire#powerrail
      Contact( "HMI_CMD_1R2".MTS_Command.SetParts."1" )
      "MTS_CreateNewPart"(II_PartType := #SI_PartType, II_DayNumber := "ProdParam".DayNumber, I_Melt := "ProdParam".Melt, XS_MatCard := "STATUS_1R2".MatCard[1, 1], XDI_PartID := #SDIPartID)
      R_Coil( "HMI_CMD_1R2".MTS_Command.SetParts."1" )
   END_RUNG
   RUNG wire#powerrail
      Contact( "HMI_CMD_1R2".MTS_Command.SetParts."2" )
      "MTS_CreateNewPart"(II_PartType := #SI_PartType, II_DayNumber := "ProdParam".DayNumber, I_Melt := "ProdParam".Melt, XS_MatCard := "STATUS_1R2".MatCard[2, 1], XDI_PartID := #SDIPartID)
      R_Coil( "HMI_CMD_1R2".MTS_Command.SetParts."2" )
   END_RUNG
   RUNG wire#powerrail
      Contact( "HMI_CMD_1R2".MTS_Command.SetParts."3" )
      "MTS_CreateNewPart"(II_PartType := #SI_PartType, II_DayNumber := "ProdParam".DayNumber, I_Melt := "ProdParam".Melt, XS_MatCard := "STATUS_1R2".MatCard[3, 1], XDI_PartID := #SDIPartID)
      R_Coil( "HMI_CMD_1R2".MTS_Command.SetParts."3" )
   END_RUNG
   RUNG wire#powerrail
      Contact( "HMI_CMD_1R2".MTS_Command.SetParts."4" )
      "MTS_CreateNewPart"(II_PartType := #SI_PartType, II_DayNumber := "ProdParam".DayNumber, I_Melt := "ProdParam".Melt, XS_MatCard := "STATUS_1R2".MatCard[4, 1], XDI_PartID := #SDIPartID)
      R_Coil( "HMI_CMD_1R2".MTS_Command.SetParts."4" )
   END_RUNG
   RUNG wire#powerrail
      Contact( "HMI_CMD_1R2".MTS_Command.SetMap )
      "MTS_MapFill"(II_PartType := #SI_PartType, X_Map := "STATUS_1R2".MatCard)
      R_Coil( "HMI_CMD_1R2".MTS_Command.SetMap )
   END_RUNG
   // the same network as SCL:
   "MTS_CreateNewPart"(EN := "HMI_CMD_1R2".MTS_Command.SetParts."1",
                       II_PartType := #SI_PartType,
                       II_DayNumber := "ProdParam".DayNumber,
                       I_Melt := "ProdParam".Melt,
                       XS_MatCard := "STATUS_1R2".MatCard[1, 1],
                       XDI_PartID := #SDIPartID,
                       ENO => #_w1);
   IF #_w1 THEN "HMI_CMD_1R2".MTS_Command.SetParts."1" := FALSE; END_IF;
   "MTS_CreateNewPart"(EN := "HMI_CMD_1R2".MTS_Command.SetParts."2",
                       II_PartType := #SI_PartType,
                       II_DayNumber := "ProdParam".DayNumber,
                       I_Melt := "ProdParam".Melt,
                       XS_MatCard := "STATUS_1R2".MatCard[2, 1],
                       XDI_PartID := #SDIPartID,
                       ENO => #_w2);
   IF #_w2 THEN "HMI_CMD_1R2".MTS_Command.SetParts."2" := FALSE; END_IF;
   "MTS_CreateNewPart"(EN := "HMI_CMD_1R2".MTS_Command.SetParts."3",
                       II_PartType := #SI_PartType,
                       II_DayNumber := "ProdParam".DayNumber,
                       I_Melt := "ProdParam".Melt,
                       XS_MatCard := "STATUS_1R2".MatCard[3, 1],
                       XDI_PartID := #SDIPartID,
                       ENO => #_w3);
   IF #_w3 THEN "HMI_CMD_1R2".MTS_Command.SetParts."3" := FALSE; END_IF;
   "MTS_CreateNewPart"(EN := "HMI_CMD_1R2".MTS_Command.SetParts."4",
                       II_PartType := #SI_PartType,
                       II_DayNumber := "ProdParam".DayNumber,
                       I_Melt := "ProdParam".Melt,
                       XS_MatCard := "STATUS_1R2".MatCard[4, 1],
                       XDI_PartID := #SDIPartID,
                       ENO => #_w4);
   IF #_w4 THEN "HMI_CMD_1R2".MTS_Command.SetParts."4" := FALSE; END_IF;
   "MTS_MapFill"(EN := "HMI_CMD_1R2".MTS_Command.SetMap,
                 II_PartType := #SI_PartType,
                 X_Map := "STATUS_1R2".MatCard,
                 ENO => #_w5);
   IF #_w5 THEN "HMI_CMD_1R2".MTS_Command.SetMap := FALSE; END_IF;
END_REGION

REGION Network 50: State evaluation of positions in gripper
   RUNG wire#powerrail
      "MTS_MapUpdateState"(IB1Clock_1s := "STDEdge_1s", X_Map := "STATUS_1R2".MatCard)
   END_RUNG
   // the same network as SCL:
   "MTS_MapUpdateState"(IB1Clock_1s := "STDEdge_1s", X_Map := "STATUS_1R2".MatCard);
END_REGION

REGION Network 51: Data transfer: 120 -> 1R2
   RUNG wire#powerrail
      Contact( "STATUS_1R2".RO01.Specific.OS_Intl.Station[1].%X2 )
      P_Trig( #SS_Edge[4] )
      "MTS_MapTakeParts"(II_RowNr := 1, II_LineNr := 1, X_Destination := "STATUS_1R2".MatCard, X_Map := "STATUS_120".MatCard)
   END_RUNG
   // the same network as SCL:
   #_w1 := "STATUS_1R2".RO01.Specific.OS_Intl.Station[1].%X2 AND NOT #SS_Edge[4];   // rising edge
   #SS_Edge[4] := "STATUS_1R2".RO01.Specific.OS_Intl.Station[1].%X2;
   IF #_w1 THEN
       "MTS_MapTakeParts"(II_RowNr := 1,
                          II_LineNr := 1,
                          X_Destination := "STATUS_1R2".MatCard,
                          X_Map := "STATUS_120".MatCard);
   END_IF;
END_REGION

REGION Network 52: Data transfer: 140 row number
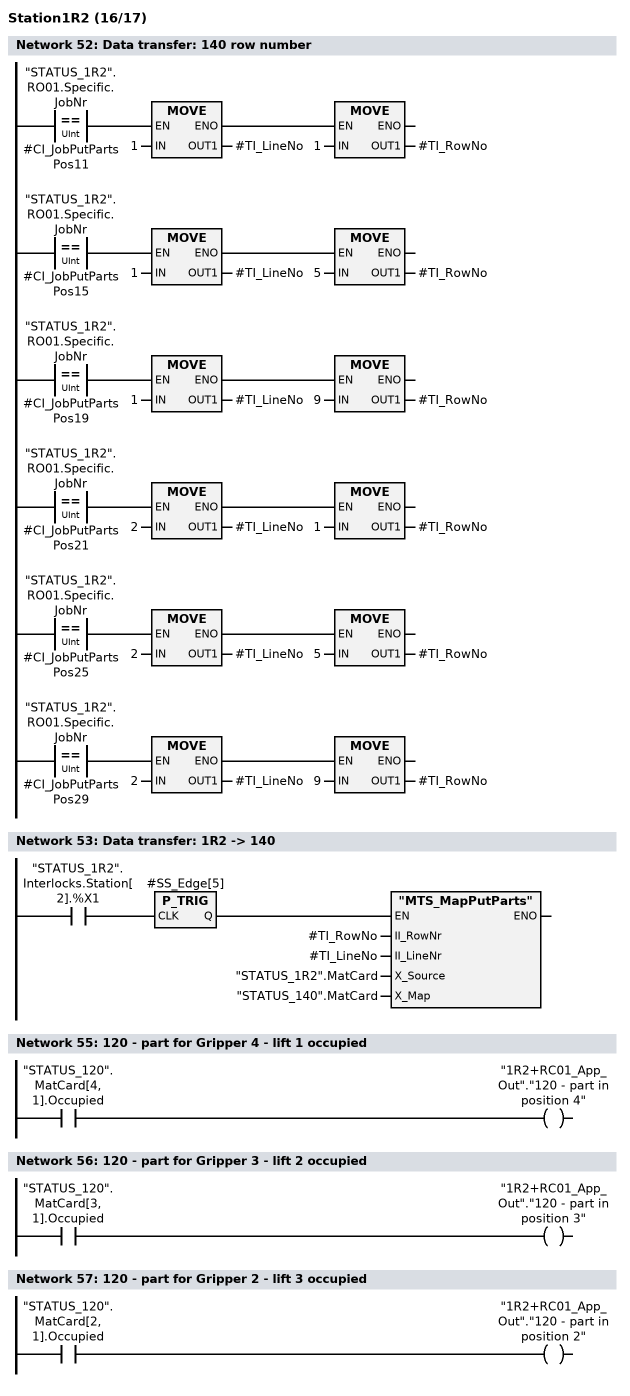
   RUNG wire#powerrail
      { S7_Templates := "SrcType := UInt" } EQ_Contact(in1 := "STATUS_1R2".RO01.Specific.JobNr, in2 := #CI_JobPutPartsPos11)
      Move(in := 1, out1 => #TI_LineNo)
      Move(in := 1, out1 => #TI_RowNo)
   END_RUNG
   RUNG wire#powerrail
      { S7_Templates := "SrcType := UInt" } EQ_Contact(in1 := "STATUS_1R2".RO01.Specific.JobNr, in2 := #CI_JobPutPartsPos15)
      Move(in := 1, out1 => #TI_LineNo)
      Move(in := 5, out1 => #TI_RowNo)
   END_RUNG
   RUNG wire#powerrail
      { S7_Templates := "SrcType := UInt" } EQ_Contact(in1 := "STATUS_1R2".RO01.Specific.JobNr, in2 := #CI_JobPutPartsPos19)
      Move(in := 1, out1 => #TI_LineNo)
      Move(in := 9, out1 => #TI_RowNo)
   END_RUNG
   RUNG wire#powerrail
      { S7_Templates := "SrcType := UInt" } EQ_Contact(in1 := "STATUS_1R2".RO01.Specific.JobNr, in2 := #CI_JobPutPartsPos21)
      Move(in := 2, out1 => #TI_LineNo)
      Move(in := 1, out1 => #TI_RowNo)
   END_RUNG
   RUNG wire#powerrail
      { S7_Templates := "SrcType := UInt" } EQ_Contact(in1 := "STATUS_1R2".RO01.Specific.JobNr, in2 := #CI_JobPutPartsPos25)
      Move(in := 2, out1 => #TI_LineNo)
      Move(in := 5, out1 => #TI_RowNo)
   END_RUNG
   RUNG wire#powerrail
      { S7_Templates := "SrcType := UInt" } EQ_Contact(in1 := "STATUS_1R2".RO01.Specific.JobNr, in2 := #CI_JobPutPartsPos29)
      Move(in := 2, out1 => #TI_LineNo)
      Move(in := 9, out1 => #TI_RowNo)
   END_RUNG
   // the same network as SCL:
   IF "STATUS_1R2".RO01.Specific.JobNr = #CI_JobPutPartsPos11 THEN
       #TI_LineNo := 1;
       #TI_RowNo := 1;
   END_IF;
   IF "STATUS_1R2".RO01.Specific.JobNr = #CI_JobPutPartsPos15 THEN
       #TI_LineNo := 1;
       #TI_RowNo := 5;
   END_IF;
   IF "STATUS_1R2".RO01.Specific.JobNr = #CI_JobPutPartsPos19 THEN
       #TI_LineNo := 1;
       #TI_RowNo := 9;
   END_IF;
   IF "STATUS_1R2".RO01.Specific.JobNr = #CI_JobPutPartsPos21 THEN
       #TI_LineNo := 2;
       #TI_RowNo := 1;
   END_IF;
   IF "STATUS_1R2".RO01.Specific.JobNr = #CI_JobPutPartsPos25 THEN
       #TI_LineNo := 2;
       #TI_RowNo := 5;
   END_IF;
   IF "STATUS_1R2".RO01.Specific.JobNr = #CI_JobPutPartsPos29 THEN
       #TI_LineNo := 2;
       #TI_RowNo := 9;
   END_IF;
END_REGION

REGION Network 53: Data transfer: 1R2 -> 140
   RUNG wire#powerrail
      Contact( "STATUS_1R2".Interlocks.Station[2].%X1 )
      P_Trig( #SS_Edge[5] )
      "MTS_MapPutParts"(II_RowNr := #TI_RowNo, II_LineNr := #TI_LineNo, X_Source := "STATUS_1R2".MatCard, X_Map := "STATUS_140".MatCard)
   END_RUNG
   // the same network as SCL:
   #_w1 := "STATUS_1R2".Interlocks.Station[2].%X1 AND NOT #SS_Edge[5];   // rising edge
   #SS_Edge[5] := "STATUS_1R2".Interlocks.Station[2].%X1;
   IF #_w1 THEN
       "MTS_MapPutParts"(II_RowNr := #TI_RowNo,
                         II_LineNr := #TI_LineNo,
                         X_Source := "STATUS_1R2".MatCard,
                         X_Map := "STATUS_140".MatCard);
   END_IF;
END_REGION

REGION Network 54: *************** Aplication Interface ***************
END_REGION

REGION Network 55: 120 - part for Gripper 4 - lift 1 occupied
   RUNG wire#powerrail
      Contact( "STATUS_120".MatCard[4, 1].Occupied )
      Coil( "1R2+RC01_App_Out"."120 - part in position 4" )
   END_RUNG
   // the same network as SCL:
   "1R2+RC01_App_Out"."120 - part in position 4" := "STATUS_120".MatCard[4, 1].Occupied;
END_REGION

REGION Network 56: 120 - part for Gripper 3 - lift 2 occupied
   RUNG wire#powerrail
      Contact( "STATUS_120".MatCard[3, 1].Occupied )
      Coil( "1R2+RC01_App_Out"."120 - part in position 3" )
   END_RUNG
   // the same network as SCL:
   "1R2+RC01_App_Out"."120 - part in position 3" := "STATUS_120".MatCard[3, 1].Occupied;
END_REGION

REGION Network 57: 120 - part for Gripper 2 - lift 3 occupied
   RUNG wire#powerrail
      Contact( "STATUS_120".MatCard[2, 1].Occupied )
      Coil( "1R2+RC01_App_Out"."120 - part in position 2" )
   END_RUNG
   // the same network as SCL:
   "1R2+RC01_App_Out"."120 - part in position 2" := "STATUS_120".MatCard[2, 1].Occupied;
END_REGION

REGION Network 58: 120 - part for Gripper 1 - lift 4 occupied
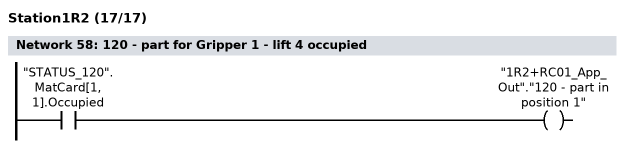
   RUNG wire#powerrail
      Contact( "STATUS_120".MatCard[1, 1].Occupied )
      Coil( "1R2+RC01_App_Out"."120 - part in position 1" )
   END_RUNG
   // the same network as SCL:
   "1R2+RC01_App_Out"."120 - part in position 1" := "STATUS_120".MatCard[1, 1].Occupied;
END_REGION
END_FUNCTION_BLOCK
